// NETWORK 70
P3_FB_Temperature[78](bReset := P3_SystemRUN.bReset, ParTemp := arrTempPar[78], TempCtrl := arrTempCtrl[78]); // FB_Temperature

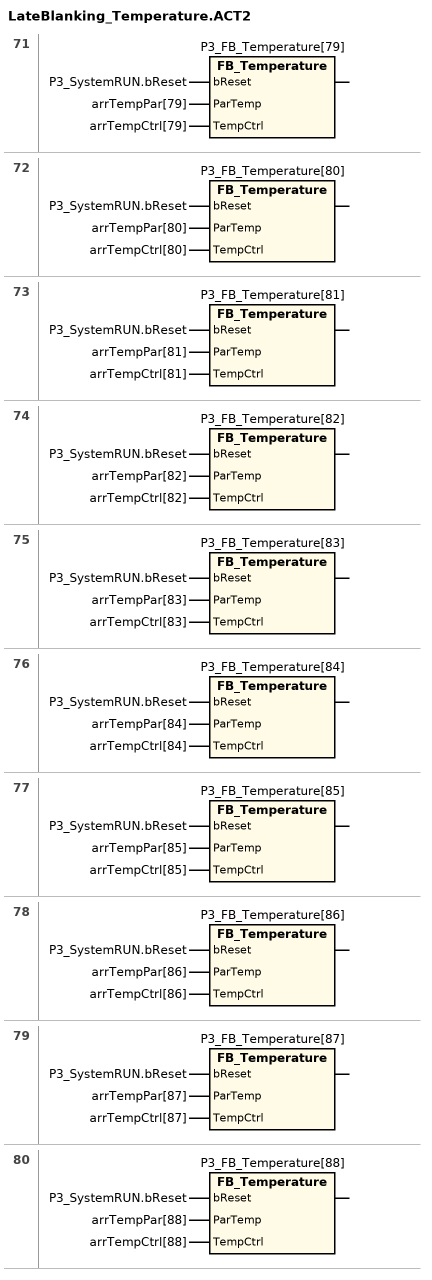
// NETWORK 71
P3_FB_Temperature[79](bReset := P3_SystemRUN.bReset, ParTemp := arrTempPar[79], TempCtrl := arrTempCtrl[79]); // FB_Temperature

// NETWORK 72
P3_FB_Temperature[80](bReset := P3_SystemRUN.bReset, ParTemp := arrTempPar[80], TempCtrl := arrTempCtrl[80]); // FB_Temperature

// NETWORK 73
P3_FB_Temperature[81](bReset := P3_SystemRUN.bReset, ParTemp := arrTempPar[81], TempCtrl := arrTempCtrl[81]); // FB_Temperature

// NETWORK 74
P3_FB_Temperature[82](bReset := P3_SystemRUN.bReset, ParTemp := arrTempPar[82], TempCtrl := arrTempCtrl[82]); // FB_Temperature

// NETWORK 75
P3_FB_Temperature[83](bReset := P3_SystemRUN.bReset, ParTemp := arrTempPar[83], TempCtrl := arrTempCtrl[83]); // FB_Temperature

// NETWORK 76
P3_FB_Temperature[84](bReset := P3_SystemRUN.bReset, ParTemp := arrTempPar[84], TempCtrl := arrTempCtrl[84]); // FB_Temperature

// NETWORK 77
P3_FB_Temperature[85](bReset := P3_SystemRUN.bReset, ParTemp := arrTempPar[85], TempCtrl := arrTempCtrl[85]); // FB_Temperature

// NETWORK 78
P3_FB_Temperature[86](bReset := P3_SystemRUN.bReset, ParTemp := arrTempPar[86], TempCtrl := arrTempCtrl[86]); // FB_Temperature

// NETWORK 79
P3_FB_Temperature[87](bReset := P3_SystemRUN.bReset, ParTemp := arrTempPar[87], TempCtrl := arrTempCtrl[87]); // FB_Temperature

// NETWORK 80
P3_FB_Temperature[88](bReset := P3_SystemRUN.bReset, ParTemp := arrTempPar[88], TempCtrl := arrTempCtrl[88]); // FB_Temperature

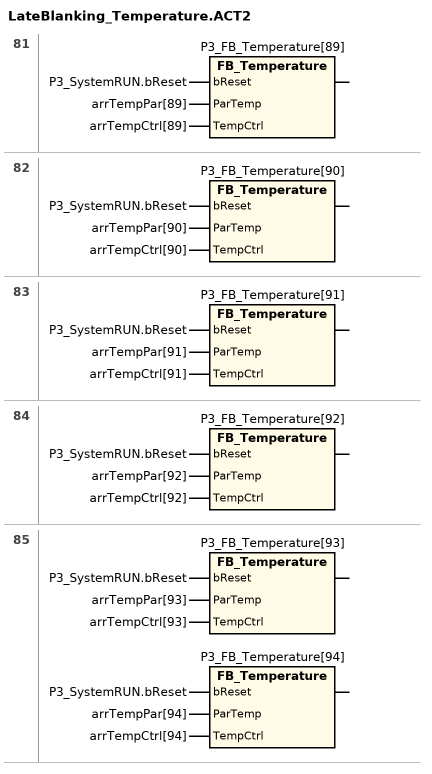
// NETWORK 81
P3_FB_Temperature[89](bReset := P3_SystemRUN.bReset, ParTemp := arrTempPar[89], TempCtrl := arrTempCtrl[89]); // FB_Temperature

// NETWORK 82
P3_FB_Temperature[90](bReset := P3_SystemRUN.bReset, ParTemp := arrTempPar[90], TempCtrl := arrTempCtrl[90]); // FB_Temperature

// NETWORK 83
P3_FB_Temperature[91](bReset := P3_SystemRUN.bReset, ParTemp := arrTempPar[91], TempCtrl := arrTempCtrl[91]); // FB_Temperature

// NETWORK 84
P3_FB_Temperature[92](bReset := P3_SystemRUN.bReset, ParTemp := arrTempPar[92], TempCtrl := arrTempCtrl[92]); // FB_Temperature

// NETWORK 85
P3_FB_Temperature[93](bReset := P3_SystemRUN.bReset, ParTemp := arrTempPar[93], TempCtrl := arrTempCtrl[93]); // FB_Temperature
P3_FB_Temperature[94](bReset := P3_SystemRUN.bReset, ParTemp := arrTempPar[94], TempCtrl := arrTempCtrl[94]); // FB_Temperature
END_ACTION

END_PROGRAM

// ---- P3POUs/POUs/Auxiliary/LateBlanking_Thickness_Test.TcPOU
//测厚测试
PROGRAM LateBlanking_Thickness_Test
VAR
b_Thickness_TON :Tc2_Standard.TON;
b_Thickness_TON2 :TON;
END_VAR

(*IF Permit_Thickness OR Shield[3]  THEN
	CellMemory[CellNo.Thickness].Thickness:=1;
    Thickness_Finish:=TRUE;
	Permit_Thickness:=FALSE;
END_IF*)
b_Thickness_TON(PT:=T#5S);
b_Thickness_TON2(PT:=T#1S);
Thickness_Par_Z:=DINT_TO_REAL(ThicknessPar)/1000;
P3User2_Par.Thick_Cell_Par:=P3User2_Par.Thick_Par - Thickness_Par_Z;
P3User2_Par.Thick_min;//:=Thick_Par-Thick_MN;
P3User2_Par.Thick_max;//:=Thick_Par+Thick_MN;

IF P3_SystemRUN.iMode=1 THEN
CASE  Thickness_Step OF

1://测厚压板打开和测厚托板缩回
	b_Thickness_TON.IN:=FALSE;
	b_Thickness_TON2.IN:=FALSE;
	IF arrCyCtrl[P3CYNo.P3ThicknessSupport].Status.ONState AND  arrCyCtrl[P3CYNo.P3ThicknessMeasuringSwitch].Status.ONState  
		AND arrCyCtrl[P3CYNo.P3ThicknessPressure].Status.OFFState THEN
		Thickness_Step:=30;
	ELSE
		Thickness_Step:=5;
	END_IF
		
5:
	arrCyCtrl[P3CYNo.P3ThicknessSupport].Cmd.bOFF:=TRUE;
	arrCyCtrl[P3CYNo.P3ThicknessPressure].Cmd.bOFF:=TRUE;
	IF 
	   arrCyCtrl[P3CYNo.P3ThicknessSupport].Status.OFFState AND NOT arrCyCtrl[P3CYNo.P3ThicknessSupport].Status.Error2 AND
	   arrCyCtrl[P3CYNo.P3ThicknessPressure].Status.OFFState AND NOT arrCyCtrl[P3CYNo.P3ThicknessPressure].Status.Error2 THEN
	   Thickness_Step:=10;
	END_IF

10://测厚切换气缸伸出
	arrCyCtrl[P3CYNo.P3ThicknessMeasuringSwitch].Cmd.bON:=TRUE;
 
	IF   arrCyCtrl[P3CYNo.P3ThicknessMeasuringSwitch].Status.ONState AND NOT arrCyCtrl[P3CYNo.P3ThicknessMeasuringSwitch].Status.Error1 THEN
		Thickness_Step:=20;
	END_IF

20://测厚托板伸出
	arrCyCtrl[P3CYNo.P3ThicknessSupport].Cmd.bON:=TRUE;
	IF 
	   arrCyCtrl[P3CYNo.P3ThicknessSupport].Status.ONState AND NOT arrCyCtrl[P3CYNo.P3ThicknessSupport].Status.Error1  THEN
	   Thickness_Step:=30;
	END_IF

30://判断是否有允许测厚信号
		IF Permit_Thickness AND NOT Thickness_Finish
		AND arrCyCtrl[P3CYNo.P3ThicknessSupport].Status.ONState AND  arrCyCtrl[P3CYNo.P3ThicknessMeasuringSwitch].Status.ONState  
		AND arrCyCtrl[P3CYNo.P3ThicknessPressure].Status.OFFState THEN
		Thickness_Step:=40;
		ELSIF Step35=100 AND(NOT arrCyCtrl[P3CYNo.P3ThicknessSupport].Status.ONState OR NOT arrCyCtrl[P3CYNo.P3ThicknessMeasuringSwitch].Status.ONState OR NOT arrCyCtrl[P3CYNo.P3ThicknessPressure].Status.OFFState) THEN
		Thickness_Step:=1;
		END_IF 
		
	
40://测厚托板缩回
	arrCyCtrl[P3CYNo.P3ThicknessSupport].Cmd.bOFF:=TRUE;
	IF 	   arrCyCtrl[P3CYNo.P3ThicknessSupport].Status.OFFState AND NOT arrCyCtrl[P3CYNo.P3ThicknessSupport].Status.Error2  THEN
	   			Thickness_Step:=50;
	END_IF  
    
50://测厚切换气缸缩回
	arrCyCtrl[P3CYNo.P3ThicknessMeasuringSwitch].Cmd.bOFF:=TRUE;
 
IF   arrCyCtrl[P3CYNo.P3ThicknessMeasuringSwitch].Status.OFFState AND NOT arrCyCtrl[P3CYNo.P3ThicknessMeasuringSwitch].Status.Error2 THEN
   Thickness_Step:=55;
END_IF

55://检测电芯有无
b_Thickness_TON2.IN:=TRUE;
IF b_Thickness_TON2.Q AND  NOT P3Senser.P3_ThicknessSensor THEN
	P3_Error[55]:=TRUE;//测厚台有记忆无电芯报警
	b_Thickness_TON2.IN:=FALSE;
	Thickness_Step:=100;
ELSE
	b_Thickness_TON2.IN:=FALSE;
	 Thickness_Step:=60;
END_IF

60://测厚压板下压
	b_Thickness_TON.IN:=FALSE;
	arrCyCtrl[P3CYNo.P3ThicknessPressure].Cmd.bON:=TRUE;
		IF    arrCyCtrl[P3CYNo.P3ThicknessPressure].Status.ONState AND NOT arrCyCtrl[P3CYNo.P3ThicknessPressure].Status.Error1 THEN
	   			Thickness_Step:=70;
		END_IF

70:
     b_Thickness_TON.IN:=TRUE;
	 IF b_Thickness_TON.Q THEN
		Thickness_Step:=80;
		b_Thickness_TON.IN:=FALSE;
	END_IF
		
80:
IF 	(P3User2_Par.Thick_Cell_Par<=P3User2_Par.Thick_max AND P3User2_Par.Thick_Cell_Par>=P3User2_Par.Thick_min) OR P3User2_Par.Shield[3] THEN
			CellMemory[CellNo.Thickness].Thickness:=1;
			CellMemory[CellNo.Thickness].Cell_Thickness:=P3User2_Par.Thick_Cell_Par;
			P3par.P3_Thickness_HMIStuas:=1;
			P3par.P3_Thickness_HMIThick:=P3User2_Par.Thick_Cell_Par;
			Thickness_Step:=90;
	ELSIF 	P3User2_Par.Thick_Cell_Par>P3User2_Par.Thick_max OR P3User2_Par.Thick_Cell_Par<P3User2_Par.Thick_min THEN
			CellMemory[CellNo.Thickness].Thickness:=2;
			CellMemory[CellNo.Thickness].Cell_Thickness:=P3User2_Par.Thick_Cell_Par;
			P3par.P3_Thickness_HMIStuas:=2;
			P3par.P3_Thickness_HMIThick:=P3User2_Par.Thick_Cell_Par;		
			Thickness_Step:=90;		
END_IF

90:
		arrCyCtrl[P3CYNo.P3ThicknessPressure].Cmd.bOFF:=TRUE;
		IF    arrCyCtrl[P3CYNo.P3ThicknessPressure].Status.OFFState AND NOT arrCyCtrl[P3CYNo.P3ThicknessPressure].Status.Error2 THEN
	   			Thickness_Step:=100;
		END_IF


100://测厚切换气缸伸出
	arrCyCtrl[P3CYNo.P3ThicknessMeasuringSwitch].Cmd.bON:=TRUE;
 
IF   arrCyCtrl[P3CYNo.P3ThicknessMeasuringSwitch].Status.ONState AND NOT arrCyCtrl[P3CYNo.P3ThicknessMeasuringSwitch].Status.Error1 THEN
   Thickness_Step:=110;
END_IF

110://测厚托板伸出
	arrCyCtrl[P3CYNo.P3ThicknessSupport].Cmd.bON:=TRUE;
	IF 
	   arrCyCtrl[P3CYNo.P3ThicknessSupport].Status.ONState AND NOT arrCyCtrl[P3CYNo.P3ThicknessSupport].Status.Error1  THEN
	   Thickness_Step:=120;
	END_IF


120:
	Permit_Thickness:=FALSE;
	Thickness_Finish:=TRUE;
	 Thickness_Step:=1;
	


		
END_CASE
END_IF

END_PROGRAM

// ---- P3POUs/POUs/Auxiliary/LateBlanking_Weight_Test.TcPOU
//称重测试
PROGRAM LateBlanking_Weight_Test
VAR
	strBetryName: STRING;//文件名

    strBetryName2: STRING;//文件名
	bTest: BOOL;
	AA: UDINT;
	BB: UDINT;
	Weight_cese_1: Weight_cese;
	
	W_ton :Tc2_Standard.TON;
	

	
END_VAR



//称重平台上料
IF NOT Permit_Weigh AND NOT Weigh_Finish THEN
	Permit_WeighRack:=TRUE;
	ELSE
	Permit_WeighRack:=FALSE;
END_IF


W_ton(PT:=T#100MS);
Weight_date();


CASE weight_step OF 
0:
IF Permit_Weigh AND NOT Weigh_Finish AND NOT P3_Error[15]THEN
	weight_step:=10;
END_IF

10:
P3_Weight_gross.Weight_start:=TRUE;
W_ton.IN:=TRUE;
weight_step:=20;

20:
IF( P3_Weight_gross.Weight_finish  AND W_ton.Q)  OR  P3User2_Par.Shield[2]	THEN
	Permit_Weigh:=FALSE;
	Weigh_Finish:=TRUE;
	P3_Weight_gross.Weight_start:=FALSE;
	CellMemory[CellNo.Weight].Cell_weight:=P3_Weight_gross.bweight;
	CellMemory[CellNo.Weight].Weight:=1;
	weight_step:=30;
END_IF

30:
W_ton.IN:=FALSE;
P3_Weight_gross.Weight_finish:=FALSE;
weight_step:=0;
END_CASE






































(*IF bTest THEN
	
 STRING_TO_UTF8(pDstUTF8:=ADR(P3WeightSend.Data) , pSrcSTRING:=ADR(strBetryName) , nDstSize:=INT_TO_UINT( LEN(STR:=strBetryName )+1) );

 AA:=INT_TO_UDINT( LEN(STR:=strBetryName2 )+1);
  BB:=INT_TO_UDINT( LEN(STR:=strBetryName )+1);
 UTF8_TO_STRING(pDstSTRING:=ADR(strBetryName2) , pSrcUTF8:=ADR(P3WeightRec.Data) , nDstSize:=SIZEOF(P3WeightRec.Data) , nDstLen=> AA    );
 bTest:=FALSE;
END_IF*)

ACTION Weight_date:
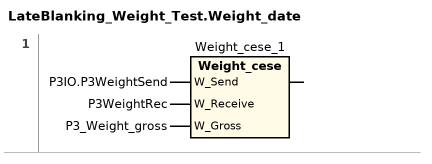
// NETWORK 1
Weight_cese_1(W_Send := P3IO.P3WeightSend, W_Receive := P3WeightRec, W_Gross := P3_Weight_gross); // Weight_cese
END_ACTION

END_PROGRAM

// ---- P3POUs/P3FB/Weight_cese.TcPOU
FUNCTION_BLOCK Weight_cese
VAR_INPUT
	//W_Send :ST_Send;
	
END_VAR
VAR_IN_OUT

	W_Send :ST_SendData;
	W_Receive:ST_ReceiveData;
	W_Gross	:ST_Gross;
END_VAR
VAR_OUTPUT
	
	
END_VAR
VAR
	Step_W_Date :UINT;
	W_TON :ARRAY[1..6] OF Tc2_Standard.TON;
	strBetryName	:STRING;//字符串
	strBetryName2 	:STRING;
	strBetryName3 	:STRING;
	L_R: UDINT;
	L_S: UDINT;
	G_OUT1 	:STRING;
	G_OUT2 	:STRING;
	weight	:REAL;
	weight_Z	:REAL;
	WeightTestAgain :BOOL;
	WeightTestAgainMount :INT;
END_VAR

ACT();
W_TON[1](PT:=T#2S);
W_TON[2](PT:=T#100MS);
W_TON[3](PT:=T#2S);
W_TON[4](PT:=T#100MS);


//初始位称重功能块
IF W_Gross.Init THEN
	Step_W_Date:=0;
	W_Gross.Weight_start:=FALSE;
	W_Gross.Clear_start:=FALSE;
	W_Send.Status.InitRequest:=FALSE;
	W_Send.Status.TransmitRequest:=FALSE;
	W_Gross.error[1]:=FALSE;
	W_Gross.Clear_finish:=FALSE;
	W_Gross.Weight_finish:=FALSE;
	W_Gross.Init:=FALSE;
END_IF





CASE Step_W_Date  OF	
0://称重测试开始
IF W_Gross.Weight_start THEN
	Step_W_Date:=10;
	W_Gross.Weight_finish:=FALSE;
	W_Gross.Weight_start :=FALSE;
	W_Gross.Clear_finish:=FALSE;

ELSIF W_Gross.Clear_start THEN
	Step_W_Date:=1010;
	W_Gross.Clear_finish:=FALSE;
	W_Gross.Clear_start :=FALSE;
	W_Gross.Weight_finish:=FALSE;
END_IF

10://初始化
W_Send.Status.InitRequest:=TRUE;
W_TON[1].IN:=TRUE;
Step_W_Date:=20;

20://如果接收到就
IF W_Receive.Status.InitAccepted THEN
	Step_W_Date:=30;
	W_Send.Status.InitRequest:=FALSE;
	W_TON[1].IN:=FALSE;
END_IF
IF W_TON[1].Q THEN
	W_Send.Status.InitRequest:=FALSE;
	W_Gross.error[1]:=TRUE;
	W_TON[1].IN:=FALSE;
	Step_W_Date:=1111;
END_IF

30:
strBetryName:='Q$R$N';
STRING_TO_UTF8(pDstUTF8:=ADR(W_Send.Data) , pSrcSTRING:=ADR(strBetryName) , nDstSize:=INT_TO_UINT( LEN(STR:=strBetryName )+1));
W_Send.Status.OutputLength:=INT_TO_UINT( LEN(STR:=strBetryName ));
Step_W_Date:=40;

40:
W_Send.Status.TransmitRequest:=TRUE;
IF W_Receive.Status.TransmitDone AND W_Receive.Status.ReceiveRequest AND W_Receive.Status.TotalInputLength>5 THEN
	Step_W_Date:=50;
W_Send.Status.TransmitRequest:=FALSE;
END_IF

50:
L_R:=INT_TO_UDINT( LEN(STR:=strBetryName2 )+1);
UTF8_TO_STRING(pDstSTRING:=ADR(strBetryName2) , pSrcUTF8:=ADR(W_Receive.Data) , nDstSize:=SIZEOF(W_Receive.Data) , nDstLen=> L_R  );
W_TON[2].IN:=TRUE;
IF W_TON[2].Q THEN
Step_W_Date:=60;
W_TON[2].IN:=FALSE;
END_IF

60:
weight_Z:=STRING_TO_REAL(G_OUT2);
IF G_OUT1='+' THEN
	W_Gross.bweight:=weight_Z;
	Step_W_Date:=70;
END_IF
IF G_OUT1='-' THEN
	W_Gross.bweight:=-weight_Z;
	Step_W_Date:=70;
END_IF

70:
IF W_Gross.bweight >=1 OR WeightTestAgain THEN
W_Gross.Weight_finish:=TRUE;
Step_W_Date:=0;
WeightTestAgain:=FALSE;
ELSE
WeightTestAgain:=TRUE;
Step_W_Date:=10;
WeightTestAgainMount:=WeightTestAgainMount+1;
END_IF




1010://初始化
W_Send.Status.InitRequest:=TRUE;
W_TON[3].IN:=TRUE;
Step_W_Date:=1020;

1020://如果接收到就
IF W_Receive.Status.InitAccepted THEN
	Step_W_Date:=1030;
	W_Send.Status.InitRequest:=FALSE;
	W_TON[3].IN:=FALSE;
END_IF
IF W_TON[3].Q THEN
	W_Send.Status.InitRequest:=FALSE;
	W_Gross.error[1]:=TRUE;
	W_TON[3].IN:=FALSE;
	Step_W_Date:=1111;
END_IF

1030:
strBetryName3:='R$R$N';
STRING_TO_UTF8(pDstUTF8:=ADR(W_Send.Data) , pSrcSTRING:=ADR(strBetryName3) , nDstSize:=INT_TO_UINT( LEN(STR:=strBetryName3 )+1   )       );
W_Send.Status.OutputLength:=INT_TO_UINT( LEN(STR:=strBetryName3 ));
Step_W_Date:=1040;

1040:
W_Send.Status.TransmitRequest:=TRUE;
IF W_Receive.Status.TransmitDone  AND W_Receive.Status.ReceiveRequest THEN
	W_Send.Status.TransmitRequest:=FALSE;
	W_Send.Status.ReceiveAccepted:=TRUE;
	Step_W_Date:=1050;
END_IF

1050:
IF NOT W_Receive.Status.ReceiveRequest  THEN
	W_Send.Status.ReceiveAccepted:=FALSE;
	Step_W_Date:=1060;
END_IF

1060:
IF  W_Receive.Status.ReceiveRequest THEN
	W_Gross.Clear_finish:=TRUE;
	Step_W_Date:=0;
END_IF



END_CASE

ACTION ACT:
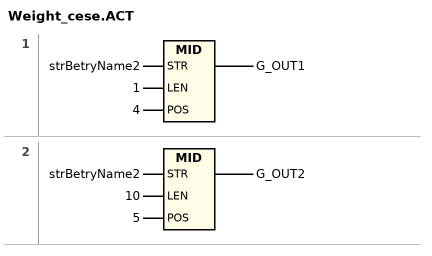
// NETWORK 1
G_OUT1 := MID(STR := strBetryName2, LEN := 1, POS := 4);

// NETWORK 2
G_OUT2 := MID(STR := strBetryName2, LEN := 10, POS := 5);
END_ACTION

END_FUNCTION_BLOCK

// ---- P3POUs/POUs/Auxiliary/LateBlankingCylinderManual.TcPOU
PROGRAM LateBlankingCylinderManual
VAR
    rGluebtn: R_TRIG;//拉胶按钮
	rCutbtn: R_TRIG;//切胶按钮
	rIDGluebtn: R_TRIG;//拉胶按钮
	rIDCutbtn: R_TRIG;//切胶按钮		
END_VAR

//冷压上料夹气缸点动
arrCyCtrl[P3CYNo.P3ColdPressClip].Cmd.ErrorTime:=5;
arrCyCtrl[P3CYNo.P3ColdPressClip].Cmd.iType:=1;
arrCyCtrl[P3CYNo.P3ColdPressClip].Cmd.OffCondition:=TRUE;
arrCyCtrl[P3CYNo.P3ColdPressClip].Cmd.OnCondition:=TRUE;

//冷压麦拉张紧气缸点动
arrCyCtrl[P3CYNo.P3ColdPressTensed].Cmd.ErrorTime:=5;
arrCyCtrl[P3CYNo.P3ColdPressTensed].Cmd.iType:=3;
arrCyCtrl[P3CYNo.P3ColdPressTensed].Cmd.OffCondition:=TRUE;
arrCyCtrl[P3CYNo.P3ColdPressTensed].Cmd.OnCondition:=TRUE;

//烤箱上料夹气缸点动
arrCyCtrl[P3CYNo.P3OvenMoveClip].Cmd.ErrorTime:=5;
arrCyCtrl[P3CYNo.P3OvenMoveClip].Cmd.iType:=1;
arrCyCtrl[P3CYNo.P3OvenMoveClip].Cmd.OffCondition:=TRUE;
arrCyCtrl[P3CYNo.P3OvenMoveClip].Cmd.OnCondition:=TRUE;


//P3 1_1烤箱托板气缸点动
arrCyCtrl[P3CYNo.P3Oven1].Cmd.ErrorTime:=8;
arrCyCtrl[P3CYNo.P3Oven1].Cmd.iType:=1;
IF arrAxisCtrlV2[P3AxisNo.P3_M2_OvenRetracting].Cmd.arrbRealPoint[43] THEN
arrCyCtrl[P3CYNo.P3Oven1].Cmd.OffCondition:=TRUE;
arrCyCtrl[P3CYNo.P3Oven1].Cmd.OnCondition:=TRUE;
ELSE
arrCyCtrl[P3CYNo.P3Oven1].Cmd.OffCondition:=FALSE;
arrCyCtrl[P3CYNo.P3Oven1].Cmd.OnCondition:=FALSE;	
END_IF

//P3 1_2烤箱托板气缸点动
arrCyCtrl[P3CYNo.P3Oven2].Cmd.ErrorTime:=7;
arrCyCtrl[P3CYNo.P3Oven2].Cmd.iType:=1;
IF arrAxisCtrlV2[P3AxisNo.P3_M2_OvenRetracting].Cmd.arrbRealPoint[43] THEN
arrCyCtrl[P3CYNo.P3Oven2].Cmd.OffCondition:=TRUE;
arrCyCtrl[P3CYNo.P3Oven2].Cmd.OnCondition:=TRUE;
ELSE
arrCyCtrl[P3CYNo.P3Oven2].Cmd.OffCondition:=FALSE;
arrCyCtrl[P3CYNo.P3Oven2].Cmd.OnCondition:=FALSE;	
END_IF


//P3 1_3烤箱托板气缸点动
arrCyCtrl[P3CYNo.P3Oven3].Cmd.ErrorTime:=7;
arrCyCtrl[P3CYNo.P3Oven3].Cmd.iType:=1;
IF arrAxisCtrlV2[P3AxisNo.P3_M2_OvenRetracting].Cmd.arrbRealPoint[43]THEN
arrCyCtrl[P3CYNo.P3Oven3].Cmd.OffCondition:=TRUE;
arrCyCtrl[P3CYNo.P3Oven3].Cmd.OnCondition:=TRUE;
ELSE
arrCyCtrl[P3CYNo.P3Oven3].Cmd.OffCondition:=FALSE;
arrCyCtrl[P3CYNo.P3Oven3].Cmd.OnCondition:=FALSE;	
END_IF

//P3 1_4烤箱托板气缸点动
arrCyCtrl[P3CYNo.P3Oven4].Cmd.ErrorTime:=7;
arrCyCtrl[P3CYNo.P3Oven4].Cmd.iType:=1;
IF arrAxisCtrlV2[P3AxisNo.P3_M2_OvenRetracting].Cmd.arrbRealPoint[43] THEN
arrCyCtrl[P3CYNo.P3Oven4].Cmd.OffCondition:=TRUE;
arrCyCtrl[P3CYNo.P3Oven4].Cmd.OnCondition:=TRUE;
ELSE
arrCyCtrl[P3CYNo.P3Oven4].Cmd.OffCondition:=FALSE;
arrCyCtrl[P3CYNo.P3Oven4].Cmd.OnCondition:=FALSE;	
END_IF

//P3 1_5烤箱托板气缸点动
arrCyCtrl[P3CYNo.P3Oven5].Cmd.ErrorTime:=7;
arrCyCtrl[P3CYNo.P3Oven5].Cmd.iType:=1;
IF arrAxisCtrlV2[P3AxisNo.P3_M2_OvenRetracting].Cmd.arrbRealPoint[43]THEN
arrCyCtrl[P3CYNo.P3Oven5].Cmd.OffCondition:=TRUE;
arrCyCtrl[P3CYNo.P3Oven5].Cmd.OnCondition:=TRUE;
ELSE
arrCyCtrl[P3CYNo.P3Oven5].Cmd.OffCondition:=FALSE;
arrCyCtrl[P3CYNo.P3Oven5].Cmd.OnCondition:=FALSE;	
END_IF

//P3 1_6烤箱托板气缸点动
arrCyCtrl[P3CYNo.P3Oven6].Cmd.ErrorTime:=7;
arrCyCtrl[P3CYNo.P3Oven6].Cmd.iType:=1;
IF arrAxisCtrlV2[P3AxisNo.P3_M2_OvenRetracting].Cmd.arrbRealPoint[43] THEN
arrCyCtrl[P3CYNo.P3Oven6].Cmd.OffCondition:=TRUE;
arrCyCtrl[P3CYNo.P3Oven6].Cmd.OnCondition:=TRUE;
ELSE
arrCyCtrl[P3CYNo.P3Oven6].Cmd.OffCondition:=FALSE;
arrCyCtrl[P3CYNo.P3Oven6].Cmd.OnCondition:=FALSE;	
END_IF

//P3 1_7烤箱托板气缸点动
arrCyCtrl[P3CYNo.P3Oven7].Cmd.ErrorTime:=7;
arrCyCtrl[P3CYNo.P3Oven7].Cmd.iType:=1;
IF arrAxisCtrlV2[P3AxisNo.P3_M2_OvenRetracting].Cmd.arrbRealPoint[43] THEN
arrCyCtrl[P3CYNo.P3Oven7].Cmd.OffCondition:=TRUE;
arrCyCtrl[P3CYNo.P3Oven7].Cmd.OnCondition:=TRUE;
ELSE
arrCyCtrl[P3CYNo.P3Oven7].Cmd.OffCondition:=FALSE;
arrCyCtrl[P3CYNo.P3Oven7].Cmd.OnCondition:=FALSE;	
END_IF

//P3 2_1烤箱托板气缸点动
arrCyCtrl[P3CYNo.P3Oven8].Cmd.ErrorTime:=7;
arrCyCtrl[P3CYNo.P3Oven8].Cmd.iType:=1;
IF arrAxisCtrlV2[P3AxisNo.P3_M2_OvenRetracting].Cmd.arrbRealPoint[43] THEN
arrCyCtrl[P3CYNo.P3Oven8].Cmd.OffCondition:=TRUE;
arrCyCtrl[P3CYNo.P3Oven8].Cmd.OnCondition:=TRUE;
ELSE
arrCyCtrl[P3CYNo.P3Oven8].Cmd.OffCondition:=FALSE;
arrCyCtrl[P3CYNo.P3Oven8].Cmd.OnCondition:=FALSE;	
END_IF

//P3 2_2烤箱托板气缸点动
arrCyCtrl[P3CYNo.P3Oven9].Cmd.ErrorTime:=7;
arrCyCtrl[P3CYNo.P3Oven9].Cmd.iType:=1;
IF arrAxisCtrlV2[P3AxisNo.P3_M2_OvenRetracting].Cmd.arrbRealPoint[43] THEN
arrCyCtrl[P3CYNo.P3Oven9].Cmd.OffCondition:=TRUE;
arrCyCtrl[P3CYNo.P3Oven9].Cmd.OnCondition:=TRUE;
ELSE
arrCyCtrl[P3CYNo.P3Oven9].Cmd.OffCondition:=FALSE;
arrCyCtrl[P3CYNo.P3Oven9].Cmd.OnCondition:=FALSE;	
END_IF

//P3 2_3烤箱托板气缸点动
arrCyCtrl[P3CYNo.P3Oven10].Cmd.ErrorTime:=7;
arrCyCtrl[P3CYNo.P3Oven10].Cmd.iType:=1;
IF arrAxisCtrlV2[P3AxisNo.P3_M2_OvenRetracting].Cmd.arrbRealPoint[43] THEN
arrCyCtrl[P3CYNo.P3Oven10].Cmd.OffCondition:=TRUE;
arrCyCtrl[P3CYNo.P3Oven10].Cmd.OnCondition:=TRUE;
ELSE
arrCyCtrl[P3CYNo.P3Oven10].Cmd.OffCondition:=FALSE;
arrCyCtrl[P3CYNo.P3Oven10].Cmd.OnCondition:=FALSE;	
END_IF

//P3 2_4烤箱托板气缸点动
arrCyCtrl[P3CYNo.P3Oven11].Cmd.ErrorTime:=7;
arrCyCtrl[P3CYNo.P3Oven11].Cmd.iType:=1;
IF arrAxisCtrlV2[P3AxisNo.P3_M2_OvenRetracting].Cmd.arrbRealPoint[43] THEN
arrCyCtrl[P3CYNo.P3Oven11].Cmd.OffCondition:=TRUE;
arrCyCtrl[P3CYNo.P3Oven11].Cmd.OnCondition:=TRUE;
ELSE
arrCyCtrl[P3CYNo.P3Oven11].Cmd.OffCondition:=FALSE;
arrCyCtrl[P3CYNo.P3Oven11].Cmd.OnCondition:=FALSE;	
END_IF

//P3 2_5烤箱托板气缸点动
arrCyCtrl[P3CYNo.P3Oven12].Cmd.ErrorTime:=7;
arrCyCtrl[P3CYNo.P3Oven12].Cmd.iType:=1;
IF arrAxisCtrlV2[P3AxisNo.P3_M2_OvenRetracting].Cmd.arrbRealPoint[43] THEN
arrCyCtrl[P3CYNo.P3Oven12].Cmd.OffCondition:=TRUE;
arrCyCtrl[P3CYNo.P3Oven12].Cmd.OnCondition:=TRUE;
ELSE
arrCyCtrl[P3CYNo.P3Oven12].Cmd.OffCondition:=FALSE;
arrCyCtrl[P3CYNo.P3Oven12].Cmd.OnCondition:=FALSE;	
END_IF

//P3 2_6烤箱托板气缸点动
arrCyCtrl[P3CYNo.P3Oven13].Cmd.ErrorTime:=7;
arrCyCtrl[P3CYNo.P3Oven13].Cmd.iType:=1;
IF arrAxisCtrlV2[P3AxisNo.P3_M2_OvenRetracting].Cmd.arrbRealPoint[43] THEN
arrCyCtrl[P3CYNo.P3Oven13].Cmd.OffCondition:=TRUE;
arrCyCtrl[P3CYNo.P3Oven13].Cmd.OnCondition:=TRUE;
ELSE
arrCyCtrl[P3CYNo.P3Oven13].Cmd.OffCondition:=FALSE;
arrCyCtrl[P3CYNo.P3Oven13].Cmd.OnCondition:=FALSE;	
END_IF

//P3 2_7烤箱托板气缸点动
arrCyCtrl[P3CYNo.P3Oven14].Cmd.ErrorTime:=7;
arrCyCtrl[P3CYNo.P3Oven14].Cmd.iType:=1;
IF arrAxisCtrlV2[P3AxisNo.P3_M2_OvenRetracting].Cmd.arrbRealPoint[43] THEN
arrCyCtrl[P3CYNo.P3Oven14].Cmd.OffCondition:=TRUE;
arrCyCtrl[P3CYNo.P3Oven14].Cmd.OnCondition:=TRUE;
ELSE
arrCyCtrl[P3CYNo.P3Oven14].Cmd.OffCondition:=FALSE;
arrCyCtrl[P3CYNo.P3Oven14].Cmd.OnCondition:=FALSE;	
END_IF

//P3 3_1烤箱托板气缸点动
arrCyCtrl[P3CYNo.P3Oven15].Cmd.ErrorTime:=7;
arrCyCtrl[P3CYNo.P3Oven15].Cmd.iType:=1;
IF arrAxisCtrlV2[P3AxisNo.P3_M2_OvenRetracting].Cmd.arrbRealPoint[43] THEN
arrCyCtrl[P3CYNo.P3Oven15].Cmd.OffCondition:=TRUE;
arrCyCtrl[P3CYNo.P3Oven15].Cmd.OnCondition:=TRUE;
ELSE
arrCyCtrl[P3CYNo.P3Oven15].Cmd.OffCondition:=FALSE;
arrCyCtrl[P3CYNo.P3Oven15].Cmd.OnCondition:=FALSE;	
END_IF

//P3 3_2烤箱托板气缸点动
arrCyCtrl[P3CYNo.P3Oven16].Cmd.ErrorTime:=7;
arrCyCtrl[P3CYNo.P3Oven16].Cmd.iType:=1;
IF arrAxisCtrlV2[P3AxisNo.P3_M2_OvenRetracting].Cmd.arrbRealPoint[43] THEN
arrCyCtrl[P3CYNo.P3Oven16].Cmd.OffCondition:=TRUE;
arrCyCtrl[P3CYNo.P3Oven16].Cmd.OnCondition:=TRUE;
ELSE
arrCyCtrl[P3CYNo.P3Oven16].Cmd.OffCondition:=FALSE;
arrCyCtrl[P3CYNo.P3Oven16].Cmd.OnCondition:=FALSE;	
END_IF

//P3 3_3烤箱托板气缸点动
arrCyCtrl[P3CYNo.P3Oven17].Cmd.ErrorTime:=7;
arrCyCtrl[P3CYNo.P3Oven17].Cmd.iType:=1;
IF arrAxisCtrlV2[P3AxisNo.P3_M2_OvenRetracting].Cmd.arrbRealPoint[43] THEN
arrCyCtrl[P3CYNo.P3Oven17].Cmd.OffCondition:=TRUE;
arrCyCtrl[P3CYNo.P3Oven17].Cmd.OnCondition:=TRUE;
ELSE
arrCyCtrl[P3CYNo.P3Oven17].Cmd.OffCondition:=FALSE;
arrCyCtrl[P3CYNo.P3Oven17].Cmd.OnCondition:=FALSE;	
END_IF

//P3 3_4烤箱托板气缸点动
arrCyCtrl[P3CYNo.P3Oven18].Cmd.ErrorTime:=7;
arrCyCtrl[P3CYNo.P3Oven18].Cmd.iType:=1;
IF arrAxisCtrlV2[P3AxisNo.P3_M2_OvenRetracting].Cmd.arrbRealPoint[43] THEN
arrCyCtrl[P3CYNo.P3Oven18].Cmd.OffCondition:=TRUE;
arrCyCtrl[P3CYNo.P3Oven18].Cmd.OnCondition:=TRUE;
ELSE
arrCyCtrl[P3CYNo.P3Oven18].Cmd.OffCondition:=FALSE;
arrCyCtrl[P3CYNo.P3Oven18].Cmd.OnCondition:=FALSE;	
END_IF

//P3 3_5烤箱托板气缸点动
arrCyCtrl[P3CYNo.P3Oven19].Cmd.ErrorTime:=7;
arrCyCtrl[P3CYNo.P3Oven19].Cmd.iType:=1;
IF arrAxisCtrlV2[P3AxisNo.P3_M2_OvenRetracting].Cmd.arrbRealPoint[43] THEN
arrCyCtrl[P3CYNo.P3Oven19].Cmd.OffCondition:=TRUE;
arrCyCtrl[P3CYNo.P3Oven19].Cmd.OnCondition:=TRUE;
ELSE
arrCyCtrl[P3CYNo.P3Oven19].Cmd.OffCondition:=FALSE;
arrCyCtrl[P3CYNo.P3Oven19].Cmd.OnCondition:=FALSE;	
END_IF

//P3 3_6烤箱托板气缸点动
arrCyCtrl[P3CYNo.P3Oven20].Cmd.ErrorTime:=7;
arrCyCtrl[P3CYNo.P3Oven20].Cmd.iType:=1;
IF arrAxisCtrlV2[P3AxisNo.P3_M2_OvenRetracting].Cmd.arrbRealPoint[43] THEN
arrCyCtrl[P3CYNo.P3Oven20].Cmd.OffCondition:=TRUE;
arrCyCtrl[P3CYNo.P3Oven20].Cmd.OnCondition:=TRUE;
ELSE
arrCyCtrl[P3CYNo.P3Oven20].Cmd.OffCondition:=FALSE;
arrCyCtrl[P3CYNo.P3Oven20].Cmd.OnCondition:=FALSE;	
END_IF

//P3 3_7烤箱托板气缸点动
arrCyCtrl[P3CYNo.P3Oven21].Cmd.ErrorTime:=7;
arrCyCtrl[P3CYNo.P3Oven21].Cmd.iType:=1;
IF arrAxisCtrlV2[P3AxisNo.P3_M2_OvenRetracting].Cmd.arrbRealPoint[43] THEN
arrCyCtrl[P3CYNo.P3Oven21].Cmd.OffCondition:=TRUE;
arrCyCtrl[P3CYNo.P3Oven21].Cmd.OnCondition:=TRUE;
ELSE
arrCyCtrl[P3CYNo.P3Oven21].Cmd.OffCondition:=FALSE;
arrCyCtrl[P3CYNo.P3Oven21].Cmd.OnCondition:=FALSE;	
END_IF

//P3 热压麦拉张紧气缸点动
arrCyCtrl[P3CYNo.P3HotPressTensed].Cmd.ErrorTime:=5;
arrCyCtrl[P3CYNo.P3HotPressTensed].Cmd.iType:=3;
arrCyCtrl[P3CYNo.P3HotPressTensed].Cmd.OffCondition:=TRUE;
arrCyCtrl[P3CYNo.P3HotPressTensed].Cmd.OnCondition:=TRUE;

//P3 短路测试夹气缸点动
arrCyCtrl[P3CYNo.P3ShortTest].Cmd.ErrorTime:=5;
arrCyCtrl[P3CYNo.P3ShortTest].Cmd.iType:=1;
arrCyCtrl[P3CYNo.P3ShortTest].Cmd.OffCondition:=TRUE;
arrCyCtrl[P3CYNo.P3ShortTest].Cmd.OnCondition:=TRUE;

//P3 称重上料夹气缸点动
arrCyCtrl[P3CYNo.P3WeightFeedingClamp].Cmd.ErrorTime:=5;
arrCyCtrl[P3CYNo.P3WeightFeedingClamp].Cmd.iType:=1;
arrCyCtrl[P3CYNo.P3WeightFeedingClamp].Cmd.OffCondition:=TRUE;
arrCyCtrl[P3CYNo.P3WeightFeedingClamp].Cmd.OnCondition:=TRUE;

//P3 测厚台切换气缸点动
arrCyCtrl[P3CYNo.P3ThicknessMeasuringSwitch].Cmd.ErrorTime:=5;
arrCyCtrl[P3CYNo.P3ThicknessMeasuringSwitch].Cmd.iType:=1;
//arrCyCtrl[P3CYNo.P3ThicknessMeasuringSwitch].Cmd.OffCondition:=TRUE;
//arrCyCtrl[P3CYNo.P3ThicknessMeasuringSwitch].Cmd.OnCondition:=TRUE;

//P3 测厚台托板气缸点动
arrCyCtrl[P3CYNo.P3ThicknessSupport].Cmd.ErrorTime:=5;
arrCyCtrl[P3CYNo.P3ThicknessSupport].Cmd.iType:=1;
//arrCyCtrl[P3CYNo.P3ThicknessSupport].Cmd.OffCondition:=TRUE;
//arrCyCtrl[P3CYNo.P3ThicknessSupport].Cmd.OnCondition:=TRUE;

//P3 测厚台压板气缸点动
arrCyCtrl[P3CYNo.P3ThicknessPressure].Cmd.ErrorTime:=5;
arrCyCtrl[P3CYNo.P3ThicknessPressure].Cmd.iType:=1;
arrCyCtrl[P3CYNo.P3ThicknessPressure].Cmd.OffCondition:=TRUE;
//arrCyCtrl[P3CYNo.P3ThicknessPressure].Cmd.OnCondition:=TRUE;

//电芯分选夹开合气缸点动
arrCyCtrl[P3CYNo.P3SortClamp].Cmd.ErrorTime:=5;
arrCyCtrl[P3CYNo.P3SortClamp].Cmd.iType:=1;
arrCyCtrl[P3CYNo.P3SortClamp].Cmd.OffCondition:=TRUE;
arrCyCtrl[P3CYNo.P3SortClamp].Cmd.OnCondition:=TRUE;

//电芯分选夹升降气缸点动
arrCyCtrl[P3CYNo.P3SortLifting].Cmd.ErrorTime:=5;
arrCyCtrl[P3CYNo.P3SortLifting].Cmd.iType:=1;
arrCyCtrl[P3CYNo.P3SortLifting].Cmd.OffCondition:=TRUE;
arrCyCtrl[P3CYNo.P3SortLifting].Cmd.OnCondition:=TRUE;

//电芯分选夹旋转气缸点动
arrCyCtrl[P3CYNo.P3SortRotate].Cmd.ErrorTime:=5;
arrCyCtrl[P3CYNo.P3SortRotate].Cmd.iType:=1;
arrCyCtrl[P3CYNo.P3SortRotate].Cmd.OffCondition:=TRUE;
arrCyCtrl[P3CYNo.P3SortRotate].Cmd.OnCondition:=TRUE;

//电芯下料夹开合气缸点动
arrCyCtrl[P3CYNo.P3BlankingClamp].Cmd.ErrorTime:=5;
arrCyCtrl[P3CYNo.P3BlankingClamp].Cmd.iType:=1;
arrCyCtrl[P3CYNo.P3BlankingClamp].Cmd.OffCondition:=TRUE;
arrCyCtrl[P3CYNo.P3BlankingClamp].Cmd.OnCondition:=TRUE;

//P3电芯下料夹升降气缸点动
arrCyCtrl[P3CYNo.P3BlankingLifting].Cmd.ErrorTime:=5;
arrCyCtrl[P3CYNo.P3BlankingLifting].Cmd.iType:=1;
arrCyCtrl[P3CYNo.P3BlankingLifting].Cmd.OffCondition:=TRUE;
arrCyCtrl[P3CYNo.P3BlankingLifting].Cmd.OnCondition:=TRUE;

//P3电芯NG1料盒锁定气缸点动
arrCyCtrl[P3CYNo.P3BoxLock1_NG].Cmd.ErrorTime:=5;
arrCyCtrl[P3CYNo.P3BoxLock1_NG].Cmd.iType:=1;
arrCyCtrl[P3CYNo.P3BoxLock1_NG].Cmd.OffCondition:=TRUE;
arrCyCtrl[P3CYNo.P3BoxLock1_NG].Cmd.OnCondition:=TRUE;

//P3电芯NG2料盒锁定气缸点动
arrCyCtrl[P3CYNo.P3BoxLock2_NG].Cmd.ErrorTime:=5;
arrCyCtrl[P3CYNo.P3BoxLock2_NG].Cmd.iType:=1;
arrCyCtrl[P3CYNo.P3BoxLock2_NG].Cmd.OffCondition:=TRUE;
arrCyCtrl[P3CYNo.P3BoxLock2_NG].Cmd.OnCondition:=TRUE;

//P3电芯NG3料盒锁定气缸点动
arrCyCtrl[P3CYNo.P3BoxLock3_NG].Cmd.ErrorTime:=5;
arrCyCtrl[P3CYNo.P3BoxLock3_NG].Cmd.iType:=1;
arrCyCtrl[P3CYNo.P3BoxLock3_NG].Cmd.OffCondition:=TRUE;
arrCyCtrl[P3CYNo.P3BoxLock3_NG].Cmd.OnCondition:=TRUE;

//电芯压紧气缸
arrCyCtrl[P3CYNo.P3CellPush].Cmd.iType:=2;

//电电芯平移气缸
arrCyCtrl[P3CYNo.P3CellAdvance].Cmd.iType:=1;

//贴胶头夹紧气缸
arrCyCtrl[P3CYNo.P3TapePush].Cmd.iType:=1;

//拉带夹紧气缸
arrCyCtrl[P3CYNo.P3TapePull].Cmd.iType:=1;

//拉带升降气缸
arrCyCtrl[P3CYNo.P3TapeLift].Cmd.iType:=1;

//切胶气缸
arrCyCtrl[P3CYNo.P3TapeCut].Cmd.iType:=1;

//压胶气缸
arrCyCtrl[P3CYNo.P3GluePush].Cmd.iType:=1;

//贴胶缓存气缸
arrCyCtrl[P3CYNo.P3TapeBuffer].Cmd.iType:=1;

//流水线下料旋转气缸
arrCyCtrl[P3CYNo.P3TapeSpin].Cmd.iType:=1;

//贴胶头真空
arrCyCtrl[P3CYNo.P3TapeVacuo].Cmd.iType:=4;


//P3称重上料夹归正气缸
arrCyCtrl[P3CYNo.P3WgightUP].Cmd.iType:=2;

//P3下料分选夹归正气缸
arrCyCtrl[P3CYNo.P3SortPush].Cmd.iType:=2;

//冷压吹气
arrCyCtrl[P3CYNo.P3ColdBlow].Cmd.iType:=4;

//热压吹气
arrCyCtrl[P3CYNo.P3HotBlow].Cmd.iType:=4;

//P3电芯旋转定位气缸 
arrCyCtrl[P3CYNo.P3CellPushSpin].Cmd.iType:=2;

//P3电芯旋转气缸
arrCyCtrl[P3CYNo.P3CellSpin].Cmd.iType:=1;


arrCyCtrl[P3CYNo.P3_GlueExtend].Cmd.iType:=4;//二维码蹬胶气缸蹬出

arrCyCtrl[P3CYNo.P3_GluePress].Cmd.iType:=2;//二维码压胶气缸压紧

arrCyCtrl[P3CYNo.P3_GlueCut].Cmd.iType:=2;//二维码切胶气缸切胶
arrCyCtrl[P3CYNo.P3_GlueCut].Cmd.OffCondition:=TRUE;
IF arrAxisCtrl[P3AxisNo.P3_IDPut].Cmd.arrbRealPoint[1] OR P3_SystemRUN.iMode=1 OR (LateBlanking_Auto1_Stick.CodeStartMark AND P3_SystemRUN.iMode=3) THEN
arrCyCtrl[P3CYNo.P3_GlueCut].Cmd.OnCondition:=TRUE;	
ELSE
arrCyCtrl[P3CYNo.P3_GlueCut].Cmd.OnCondition:=FALSE;	
END_IF


arrCyCtrl[P3CYNo.P3_GluePull].Cmd.iType:=2;//二维码拉胶气缸夹紧

arrCyCtrl[P3CYNo.P3_GlueVacuum].Cmd.iType:=4;//	二维码贴胶吸盘真空






//拉胶气缸手动
rGluebtn(CLK:=P3Press.Gluebtn , Q=> );
IF NOT arrCyCtrl[P3CYNo.P3TapeLift].Status.OFFState AND rGluebtn.Q AND P3_SystemRUN.iMode=3 AND arrAxisCtrl[P3AxisNo.P3_TapeAdvance].Cmd.arrbRealPoint[1]  
  (* LREAL_TO_REAL(arrAxisCtrl[P3AxisNo.P3_TapeAdvance].Status.fActPos) <= (arrAxisPar[P3AxisNo.P3_TapeAdvance].arrTargetPoint[1]+1)*) THEN
	arrCyCtrl[P3CYNo.P3TapeLift].Cmd.bOFF:=TRUE;
ELSIF NOT arrCyCtrl[P3CYNo.P3TapeLift].Status.ONState AND rGluebtn.Q AND P3_SystemRUN.iMode=3 AND arrAxisCtrl[P3AxisNo.P3_TapeAdvance].Cmd.arrbRealPoint[1]  AND
          arrCyCtrl[P3CYNo.P3TapeCut].Status.OFFState  THEN
	arrCyCtrl[P3CYNo.P3TapeLift].Cmd.bON:=TRUE;
END_IF

//切胶气缸手动
rCutbtn(CLK:=P3Press.Cutbtn , Q=> );
IF NOT arrCyCtrl[P3CYNo.P3TapeCut].Status.OFFState AND rCutbtn.Q AND P3_SystemRUN.iMode=3 THEN
	arrCyCtrl[P3CYNo.P3TapeCut].Cmd.bOFF:=TRUE;
ELSIF NOT arrCyCtrl[P3CYNo.P3TapeCut].Status.ONState AND rCutbtn.Q AND P3_SystemRUN.iMode=3 AND
      arrCyCtrl[P3CYNo.P3TapeLift].Status.OFFState THEN
	arrCyCtrl[P3CYNo.P3TapeCut].Cmd.bON:=TRUE;
END_IF
//切胶气缸手动
rIDCutbtn(CLK:=P3Button.IDCutbtn , Q=> );
IF NOT arrCyCtrl[P3CYNo.P3_GlueCut].Status.OFFState AND rIDCutbtn.Q AND P3_SystemRUN.iMode=3 THEN
	arrCyCtrl[P3CYNo.P3_GlueCut].Cmd.bOFF:=TRUE;
ELSIF NOT arrCyCtrl[P3CYNo.P3_GlueCut].Status.ONState AND rIDCutbtn.Q AND P3_SystemRUN.iMode=3 THEN
	arrCyCtrl[P3CYNo.P3_GlueCut].Cmd.bON:=TRUE;
END_IF

END_PROGRAM

// ---- P3POUs/POUs/Auxiliary/LateBlankingMotorManual.TcPOU
PROGRAM LateBlankingMotorManual
VAR
END_VAR

(*//P3_M1冷压上料夹平移点动
IF arrAxisCtrl[P3AxisNo.P3M1_ColdpreLine].Cmd.hmiJog_Fw THEN
arrAxisCtrl[P3AxisNo.P3M1_ColdpreLine].Cmd.bJog_Fw:=TRUE;
ELSE
arrAxisCtrl[P3AxisNo.P3M1_ColdpreLine].Cmd.bJog_Fw:=FALSE;
END_IF
IF arrAxisCtrl[P3AxisNo.P3M1_ColdpreLine].Cmd.hmibJog_Bw THEN
arrAxisCtrl[P3AxisNo.P3M1_ColdpreLine].Cmd.bJog_Bw:=TRUE;
ELSE
arrAxisCtrl[P3AxisNo.P3M1_ColdpreLine].Cmd.bJog_Bw:=FALSE;
END_IF

//P3_M1冷压上料夹进退点动
IF arrAxisCtrl[P3AxisNo.P3M1_ColdpreRetracting].Cmd.hmiJog_Fw THEN
arrAxisCtrl[P3AxisNo.P3M1_ColdpreRetracting].Cmd.bJog_Fw:=TRUE;
ELSE
arrAxisCtrl[P3AxisNo.P3M1_ColdpreRetracting].Cmd.bJog_Fw:=FALSE;
END_IF
IF arrAxisCtrl[P3AxisNo.P3M1_ColdpreRetracting].Cmd.hmibJog_Bw THEN
arrAxisCtrl[P3AxisNo.P3M1_ColdpreRetracting].Cmd.bJog_Bw:=TRUE;
ELSE
arrAxisCtrl[P3AxisNo.P3M1_ColdpreRetracting].Cmd.bJog_Bw:=FALSE;
END_IF

//P3_M1冷压上料夹旋转点动
IF arrAxisCtrl[P3AxisNo.P3M1_ColdpreWhirling].Cmd.hmiJog_Fw THEN
arrAxisCtrl[P3AxisNo.P3M1_ColdpreWhirling].Cmd.bJog_Fw:=TRUE;
ELSE
arrAxisCtrl[P3AxisNo.P3M1_ColdpreWhirling].Cmd.bJog_Fw:=FALSE;
END_IF
IF arrAxisCtrl[P3AxisNo.P3M1_ColdpreWhirling].Cmd.hmibJog_Bw THEN
arrAxisCtrl[P3AxisNo.P3M1_ColdpreWhirling].Cmd.bJog_Bw:=TRUE;
ELSE
arrAxisCtrl[P3AxisNo.P3M1_ColdpreWhirling].Cmd.bJog_Bw:=FALSE;
END_IF

//P3_M1冷压上料夹升降点动
IF arrAxisCtrl[P3AxisNo.P3M1_ColdpreUpDown].Cmd.hmiJog_Fw THEN
arrAxisCtrl[P3AxisNo.P3M1_ColdpreUpDown].Cmd.bJog_Fw:=TRUE;
ELSE
arrAxisCtrl[P3AxisNo.P3M1_ColdpreUpDown].Cmd.bJog_Fw:=FALSE;
END_IF
IF arrAxisCtrl[P3AxisNo.P3M1_ColdpreUpDown].Cmd.hmibJog_Bw THEN
arrAxisCtrl[P3AxisNo.P3M1_ColdpreUpDown].Cmd.bJog_Bw:=TRUE;
ELSE
arrAxisCtrl[P3AxisNo.P3M1_ColdpreUpDown].Cmd.bJog_Bw:=FALSE;
END_IF

//P3_M1冷压托板开合点动
IF arrAxisCtrl[P3AxisNo.P3M1_ColdpreSupPlateLine].Cmd.hmiJog_Fw THEN
arrAxisCtrl[P3AxisNo.P3M1_ColdpreSupPlateLine].Cmd.bJog_Fw:=TRUE;
ELSE
arrAxisCtrl[P3AxisNo.P3M1_ColdpreSupPlateLine].Cmd.bJog_Fw:=FALSE;
END_IF
IF arrAxisCtrl[P3AxisNo.P3M1_ColdpreSupPlateLine].Cmd.hmibJog_Bw THEN
arrAxisCtrl[P3AxisNo.P3M1_ColdpreSupPlateLine].Cmd.bJog_Bw:=TRUE;
ELSE
arrAxisCtrl[P3AxisNo.P3M1_ColdpreSupPlateLine].Cmd.bJog_Bw:=FALSE;
END_IF

//P3_M1冷压驱动点动
IF arrAxisCtrl[P3AxisNo.P3M1_ColdpreActuated].Cmd.hmiJog_Fw THEN
arrAxisCtrl[P3AxisNo.P3M1_ColdpreActuated].Cmd.bJog_Fw:=TRUE;
ELSE
arrAxisCtrl[P3AxisNo.P3M1_ColdpreActuated].Cmd.bJog_Fw:=FALSE;
END_IF
IF arrAxisCtrl[P3AxisNo.P3M1_ColdpreActuated].Cmd.hmibJog_Bw THEN
arrAxisCtrl[P3AxisNo.P3M1_ColdpreActuated].Cmd.bJog_Bw:=TRUE;
ELSE
arrAxisCtrl[P3AxisNo.P3M1_ColdpreActuated].Cmd.bJog_Bw:=FALSE;
END_IF

//P3_M2烤箱上料夹搬运点动
IF arrAxisCtrlV2[P3AxisNo.P3_M2_OvenCarrying].Cmd.hmiJog_Fw THEN
arrAxisCtrlV2[P3AxisNo.P3_M2_OvenCarrying].Cmd.bJog_Fw:=TRUE;
ELSE
arrAxisCtrlV2[P3AxisNo.P3_M2_OvenCarrying].Cmd.bJog_Fw:=FALSE;
END_IF
IF arrAxisCtrlV2[P3AxisNo.P3_M2_OvenCarrying].Cmd.hmibJog_Bw THEN
arrAxisCtrlV2[P3AxisNo.P3_M2_OvenCarrying].Cmd.bJog_Bw:=TRUE;
ELSE
arrAxisCtrlV2[P3AxisNo.P3_M2_OvenCarrying].Cmd.bJog_Bw:=FALSE;
END_IF

//P3_M2烤箱上料夹进退点动
IF arrAxisCtrlV2[P3AxisNo.P3_M2_OvenRetracting].Cmd.hmiJog_Fw THEN
arrAxisCtrlV2[P3AxisNo.P3_M2_OvenRetracting].Cmd.bJog_Fw:=TRUE;
ELSE
arrAxisCtrlV2[P3AxisNo.P3_M2_OvenRetracting].Cmd.bJog_Fw:=FALSE;
END_IF
IF arrAxisCtrlV2[P3AxisNo.P3_M2_OvenRetracting].Cmd.hmibJog_Bw THEN
arrAxisCtrlV2[P3AxisNo.P3_M2_OvenRetracting].Cmd.bJog_Bw:=TRUE;
ELSE
arrAxisCtrlV2[P3AxisNo.P3_M2_OvenRetracting].Cmd.bJog_Bw:=FALSE;
END_IF

//P3_M2烤箱上料夹升降点动
IF arrAxisCtrlV2[P3AxisNo.P3_M2_OvenUpDown].Cmd.hmiJog_Fw THEN
arrAxisCtrlV2[P3AxisNo.P3_M2_OvenUpDown].Cmd.bJog_Fw:=TRUE;
ELSE
arrAxisCtrlV2[P3AxisNo.P3_M2_OvenUpDown].Cmd.bJog_Fw:=FALSE;
END_IF
IF arrAxisCtrlV2[P3AxisNo.P3_M2_OvenUpDown].Cmd.hmibJog_Bw THEN
arrAxisCtrlV2[P3AxisNo.P3_M2_OvenUpDown].Cmd.bJog_Bw:=TRUE;
ELSE
arrAxisCtrlV2[P3AxisNo.P3_M2_OvenUpDown].Cmd.bJog_Bw:=FALSE;
END_IF

//P3_M3热压托板开合点动
IF arrAxisCtrl[P3AxisNo.P3_M3_HotPressingLine].Cmd.hmiJog_Fw THEN
arrAxisCtrl[P3AxisNo.P3_M3_HotPressingLine].Cmd.bJog_Fw:=TRUE;
ELSE
arrAxisCtrl[P3AxisNo.P3_M3_HotPressingLine].Cmd.bJog_Fw:=FALSE;
END_IF
IF arrAxisCtrl[P3AxisNo.P3_M3_HotPressingLine].Cmd.hmibJog_Bw THEN
arrAxisCtrl[P3AxisNo.P3_M3_HotPressingLine].Cmd.bJog_Bw:=TRUE;
ELSE
arrAxisCtrl[P3AxisNo.P3_M3_HotPressingLine].Cmd.bJog_Bw:=FALSE;
END_IF

//P3_M3热压驱动点动
IF arrAxisCtrl[P3AxisNo.P3_M3_HotPressingActuated].Cmd.hmiJog_Fw THEN
arrAxisCtrl[P3AxisNo.P3_M3_HotPressingActuated].Cmd.bJog_Fw:=TRUE;
ELSE
arrAxisCtrl[P3AxisNo.P3_M3_HotPressingActuated].Cmd.bJog_Fw:=FALSE;
END_IF
IF arrAxisCtrl[P3AxisNo.P3_M3_HotPressingActuated].Cmd.hmibJog_Bw THEN
arrAxisCtrl[P3AxisNo.P3_M3_HotPressingActuated].Cmd.bJog_Bw:=TRUE;
ELSE
arrAxisCtrl[P3AxisNo.P3_M3_HotPressingActuated].Cmd.bJog_Bw:=FALSE;
END_IF

//P3_M4称重上料夹平移点动
IF arrAxisCtrl[P3AxisNo.P3_M4_WeighLine].Cmd.hmiJog_Fw THEN
arrAxisCtrl[P3AxisNo.P3_M4_WeighLine].Cmd.bJog_Fw:=TRUE;
ELSE
arrAxisCtrl[P3AxisNo.P3_M4_WeighLine].Cmd.bJog_Fw:=FALSE;
END_IF
IF arrAxisCtrl[P3AxisNo.P3_M4_WeighLine].Cmd.hmibJog_Bw THEN
arrAxisCtrl[P3AxisNo.P3_M4_WeighLine].Cmd.bJog_Bw:=TRUE;
ELSE
arrAxisCtrl[P3AxisNo.P3_M4_WeighLine].Cmd.bJog_Bw:=FALSE;
END_IF

//P3_M4称重上料夹升降点动
IF arrAxisCtrl[P3AxisNo.P3_M4_WeighUpDown].Cmd.hmiJog_Fw THEN
arrAxisCtrl[P3AxisNo.P3_M4_WeighUpDown].Cmd.bJog_Fw:=TRUE;
ELSE
arrAxisCtrl[P3AxisNo.P3_M4_WeighUpDown].Cmd.bJog_Fw:=FALSE;
END_IF
IF arrAxisCtrl[P3AxisNo.P3_M4_WeighUpDown].Cmd.hmibJog_Bw THEN
arrAxisCtrl[P3AxisNo.P3_M4_WeighUpDown].Cmd.bJog_Bw:=TRUE;
ELSE
arrAxisCtrl[P3AxisNo.P3_M4_WeighUpDown].Cmd.bJog_Bw:=FALSE;
END_IF

//P3_M4称重上料夹旋转点动
IF arrAxisCtrl[P3AxisNo.P3_M4_WeighWhirling].Cmd.hmiJog_Fw THEN
arrAxisCtrl[P3AxisNo.P3_M4_WeighWhirling].Cmd.bJog_Fw:=TRUE;
ELSE
arrAxisCtrl[P3AxisNo.P3_M4_WeighWhirling].Cmd.bJog_Fw:=FALSE;
END_IF
IF arrAxisCtrl[P3AxisNo.P3_M4_WeighWhirling].Cmd.hmibJog_Bw THEN
arrAxisCtrl[P3AxisNo.P3_M4_WeighWhirling].Cmd.bJog_Bw:=TRUE;
ELSE
arrAxisCtrl[P3AxisNo.P3_M4_WeighWhirling].Cmd.bJog_Bw:=FALSE;
END_IF

//P3_M4电芯分选夹搬运点动
IF arrAxisCtrl[P3AxisNo.P3_M4_SortingoutCarrying].Cmd.hmiJog_Fw THEN
arrAxisCtrl[P3AxisNo.P3_M4_SortingoutCarrying].Cmd.bJog_Fw:=TRUE;
ELSE
arrAxisCtrl[P3AxisNo.P3_M4_SortingoutCarrying].Cmd.bJog_Fw:=FALSE;
END_IF
IF arrAxisCtrl[P3AxisNo.P3_M4_SortingoutCarrying].Cmd.hmibJog_Bw THEN
arrAxisCtrl[P3AxisNo.P3_M4_SortingoutCarrying].Cmd.bJog_Bw:=TRUE;
ELSE
arrAxisCtrl[P3AxisNo.P3_M4_SortingoutCarrying].Cmd.bJog_Bw:=FALSE;
END_IF

//P3_M4电芯分选夹升降点动
IF arrAxisCtrl[P3AxisNo.P3_M4_SortingoutUpDown].Cmd.hmiJog_Fw THEN
arrAxisCtrl[P3AxisNo.P3_M4_SortingoutUpDown].Cmd.bJog_Fw:=TRUE;
ELSE
arrAxisCtrl[P3AxisNo.P3_M4_SortingoutUpDown].Cmd.bJog_Fw:=FALSE;
END_IF
IF arrAxisCtrl[P3AxisNo.P3_M4_SortingoutUpDown].Cmd.hmibJog_Bw THEN
arrAxisCtrl[P3AxisNo.P3_M4_SortingoutUpDown].Cmd.bJog_Bw:=TRUE;
ELSE
arrAxisCtrl[P3AxisNo.P3_M4_SortingoutUpDown].Cmd.bJog_Bw:=FALSE;
END_IF

//P3_M4电芯下料夹搬运点动
IF arrAxisCtrl[P3AxisNo.P3_M4_OffloadingCarrying].Cmd.hmiJog_Fw THEN
arrAxisCtrl[P3AxisNo.P3_M4_OffloadingCarrying].Cmd.bJog_Fw:=TRUE;
ELSE
arrAxisCtrl[P3AxisNo.P3_M4_OffloadingCarrying].Cmd.bJog_Fw:=FALSE;
END_IF
IF arrAxisCtrl[P3AxisNo.P3_M4_OffloadingCarrying].Cmd.hmibJog_Bw THEN
arrAxisCtrl[P3AxisNo.P3_M4_OffloadingCarrying].Cmd.bJog_Bw:=TRUE;
ELSE
arrAxisCtrl[P3AxisNo.P3_M4_OffloadingCarrying].Cmd.bJog_Bw:=FALSE;
END_IF

//P3_M4电芯下料夹升降点动
IF arrAxisCtrl[P3AxisNo.P3_M4_OffloadingUpDown].Cmd.hmiJog_Fw THEN
arrAxisCtrl[P3AxisNo.P3_M4_OffloadingUpDown].Cmd.bJog_Fw:=TRUE;
ELSE
arrAxisCtrl[P3AxisNo.P3_M4_OffloadingUpDown].Cmd.bJog_Fw:=FALSE;
END_IF
IF arrAxisCtrl[P3AxisNo.P3_M4_OffloadingUpDown].Cmd.hmibJog_Bw THEN
arrAxisCtrl[P3AxisNo.P3_M4_OffloadingUpDown].Cmd.bJog_Bw:=TRUE;
ELSE
arrAxisCtrl[P3AxisNo.P3_M4_OffloadingUpDown].Cmd.bJog_Bw:=FALSE;
END_IF
*)

END_PROGRAM

// ---- P3POUs/POUs/Auxiliary/LateBlanking_Short_Test.TcPOU
PROGRAM LateBlanking_Short_Test
VAR
ShortTest_Start_TON :Tc2_Standard.TON;	
TON_CYShort :Tc2_Standard.TON;
ShortTest_0: ShortTest;
Shortdata_ton :Tc2_Standard.TON;
YS_Short_ton :Tc2_Standard.TON;
FC_ton :Tc2_Standard.TON;
I:INT;
NG_Tim:Tc2_Standard.TON;
OK_Tim:Tc2_Standard.TON;
END_VAR

(*//短路测试//////////////////开通短路测试要删掉
IF Permit_ShortTest OR Shield[1] THEN
	CellMemory[CellNo.Hotpress].ShortTest:=1;
	ShortTest_Finish:=TRUE;
	Permit_ShortTest:=FALSE;
END_IF*)
shortcese();
ShortTest_Start_TON(PT:=T#8S);
TON_CYShort(PT:=T#6S);
Shortdata_ton(PT:=T#200MS);
YS_Short_ton(PT:=T#3.5S);
FC_ton(PT:=T#70MS);



//IF P3_SystemRUN.iMode=1  THEN//OR P3_SystemRUN.iMode=3
CASE Step_Short OF
0:
	TON_CYShort.IN:=FALSE;
	ShortTest_Start_TON.IN:=FALSE;
	arrCyCtrl[P3CYNo.P3ShortTest].Cmd.bOFF:=TRUE;
	P3Senser.P3_ShortTest_Start:=FALSE;
	Shortdata_ton.IN:=FALSE;
	YS_Short_ton.IN:=FALSE;	
	FC_ton.IN:=FALSE;
	I:=0;
	IF arrCyCtrl[P3CYNo.P3ShortTest].Status.OFFState AND NOT arrCyCtrl[P3CYNo.P3ShortTest].Status.Error2   THEN	
		Step_Short:=5;
	END_IF
5:
	IF  NOT ShortTest_Finish AND Permit_ShortTest AND arrAxisCtrl[P3AxisNo.P3_M3_HotPressingLine].Cmd.arrbRealPoint[2]
		 AND arrAxisCtrl[P3AxisNo.P3_M3_HotPressingLine].Status.NoMoving THEN
		Step_Short:=10;
	END_IF
10:
	IF P3User2_Par.Shield[1] THEN
		Step_Short:=0;
		ShortTest_Finish:=TRUE;	
		CellMemory[CellNo.Hotpress].ShortTest:=1;
	ELSIF Permit_ShortTest AND NOT ShortTest_Finish AND NOT P3Senser.P3_ShortTest_Testing AND Pressing[2] THEN
		 Step_Short:=20;
	END_IF 

20:
	TON_CYShort.IN:=TRUE;
    arrCyCtrl[P3CYNo.P3ShortTest].Cmd.bON:=TRUE;	
	IF (arrCyCtrl[P3CYNo.P3ShortTest].Status.ONState AND NOT arrCyCtrl[P3CYNo.P3ShortTest].Status.Error1) OR TON_CYShort.Q THEN	
	Step_Short:=30;
	TON_CYShort.IN:=FALSE;
	END_IF
		
30:
TON_CYShort.IN:=FALSE;
ShortTest_Start_TON.IN:=TRUE;
P3Senser.P3_ShortTest_Start:=TRUE;
IF ShortTest_Start_TON.Q THEN
Step_Short:=40;
ShortTest_Start_TON.IN:=FALSE;
END_IF

40:
ShortTest_Start_TON.IN:=FALSE;
Shortdata_ton.IN:=FALSE;
OK_Tim(IN:=P3Senser.P3_ShortTest_Pass , PT:=T#0.5S , Q=> , ET=> );
NG_Tim(IN:=P3Senser.P3_ShortTest_UpperFall OR P3Senser.P3_ShortTest_LowerFall , PT:=T#0.5S , Q=> , ET=> );
IF NG_Tim.Q THEN
//IF P3Senser.P3_ShortTest_UpperFall OR P3Senser.P3_ShortTest_LowerFall THEN
	CellMemory[CellNo.Hotpress].ShortTest:=2;
	NG_Tim(IN:=FALSE );
	Step_Short:=50;
	SHORT_HOT.bStart:=TRUE;
ELSIF OK_Tim.Q THEN
//ELSIF P3Senser.P3_ShortTest_Pass THEN
	CellMemory[CellNo.Hotpress].ShortTest:=1;
	OK_Tim(IN:=FALSE );
	Step_Short:=50;
	SHORT_HOT.bStart:=TRUE;	
END_IF

50:
Shortdata_ton.IN:=TRUE;
IF Shortdata_ton.Q AND SHORT_HOT.bDone THEN
Step_Short:=60;	
Shortdata_ton.IN:=FALSE;
END_IF

60:
CellMemory[CellNo.Hotpress].Hipot_R:=(SHORT_HOT.Measure);
CellMemory[CellNo.Hotpress].Hipot_Time:=SHORT_HOT.TestTime;
CellMemory[CellNo.Hotpress].Hipot_V:=SHORT_HOT.Voltage;
Step_Short:=70;	

70:
FC_ton.IN:=FALSE;
SHORT_HOT.bDone:=FALSE;
YS_Short_ton.IN:=FALSE;
P3Senser.P3_ShortTest_Start:=FALSE;
arrCyCtrl[P3CYNo.P3ShortTest].Cmd.bOFF:=TRUE;
Step_Short:=73;	

73:
IF ((CellMemory[CellNo.Hotpress].Hipot_R=0 AND CellMemory[CellNo.Hotpress].ShortTest<>2) 
OR CellMemory[CellNo.Hotpress].Hipot_Time=0 OR CellMemory[CellNo.Hotpress].Hipot_V=0) AND I<=3 THEN
	Step_Short:=1000;

	ELSIF ((CellMemory[CellNo.Hotpress].Hipot_R=0 AND CellMemory[CellNo.Hotpress].ShortTest<>2) 
OR CellMemory[CellNo.Hotpress].Hipot_Time=0 OR CellMemory[CellNo.Hotpress].Hipot_V=0) AND I>3 THEN
	Step_Short:=75;
	I:=0;
	CellMemory[CellNo.Hotpress].Hipot_R:=0;
	CellMemory[CellNo.Hotpress].ShortTest:=2;
	ELSE
	Step_Short:=75;
END_IF

(*
75:
	ShortTest_Finish:=TRUE;
	Permit_ShortTest:=FALSE;
	Step_Short:=0;	*)
75:
	IF NOT P3User2_Par.Shield[6] OR CellMemory[CellNo.Hotpress].ShortTest=2 THEN
		ShortTest_Finish:=TRUE;
		Permit_ShortTest:=FALSE;
		Step_Short:=0;	
	ELSE
	   Step_Short:=80;		
	END_IF



80:
YS_Short_ton.IN:=TRUE;	
IF YS_Short_ton.Q THEN
	arrCyCtrl[P3CYNo.P3ShortTest].Cmd.bON:=TRUE;
	YS_Short_ton.IN:=FALSE;
	TON_CYShort.IN:=TRUE;
	Step_Short:=90;
END_IF

90:
	IF TON_CYShort.Q THEN
		ShortTest_Start_TON.IN:=TRUE;
		P3Senser.P3_ShortTest_Start:=TRUE;
		TON_CYShort.IN:=FALSE;
		Step_Short:=100;
	END_IF
	
100:
	IF ShortTest_Start_TON.Q THEN
		Step_Short:=110;
		SHORT_HOT.bStart:=TRUE;
		ShortTest_Start_TON.IN:=FALSE;
	END_IF

110:
  IF P3Senser.P3_ShortTest_Pass AND CellMemory[CellNo.Hotpress].ShortTest=1 THEN
	  CellMemory[CellNo.Hotpress].ShortTest:=1;
	  Step_Short:=120;
	  ELSIF P3Senser.P3_ShortTest_UpperFall OR P3Senser.P3_ShortTest_LowerFall THEN
	   CellMemory[CellNo.Hotpress].ShortTest:=2;
	    Step_Short:=120;
  END_IF

120:
Shortdata_ton.IN:=TRUE;
IF Shortdata_ton.Q AND SHORT_HOT.bDone THEN
Step_Short:=130;	
Shortdata_ton.IN:=FALSE;
END_IF

130:
CellMemory[CellNo.Hotpress].Hipot2_R:=SHORT_HOT.Measure;
Step_Short:=140;	

140:
SHORT_HOT.bDone:=FALSE;
YS_Short_ton.IN:=FALSE;
P3Senser.P3_ShortTest_Start:=FALSE;
arrCyCtrl[P3CYNo.P3ShortTest].Cmd.bOFF:=TRUE;
ShortTest_Finish:=TRUE;
Permit_ShortTest:=FALSE;
Step_Short:=0;	
	
1000:
SHORT_HOT.bStart:=TRUE;
FC_ton.IN:=TRUE;
Step_Short:=1010;

1010:
IF  SHORT_HOT.bDone AND FC_ton.Q THEN
Step_Short:=60;	
FC_ton.IN:=FALSE;
I:=I+1;
END_IF



	
	
END_CASE
//END_IF

ACTION shortcese:
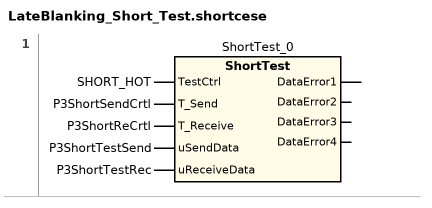
// NETWORK 1
ShortTest_0(
    TestCtrl := SHORT_HOT,
    T_Send := P3ShortSendCrtl,
    T_Receive := P3ShortReCrtl,
    uSendData := P3ShortTestSend,
    uReceiveData := P3ShortTestRec); // ShortTest
END_ACTION

END_PROGRAM

// ---- P3POUs/POUs/Auxiliary/LateBlanking_Scan.TcPOU
PROGRAM LateBlanking_Scan
VAR
	CS_CodeTcp_cold: CS_CodeTcp;
	Cold_step :UINT;
	scan_TON1 :Tc2_Standard.TON;
	Scan_TON :ARRAY[1..7] OF Tc2_Standard.TON;
	Scan_code_Z : R_TRIG;
	I:INT;
END_VAR

//扫码



Saoma();
P3User2_Par.Scan_IP:='192.168.10.26';
Scan_TON[1](PT:=T#1MS);
Scan_TON[2](PT:=T#1MS);
Scan_TON[3](PT:=T#1MS);
Scan_TON[4](PT:=T#100MS);

Scan_code_Z (CLK:=Cold_Scan_code, Q=>);

IF Scan_code_Z.Q AND  Cold_step=0 THEN
	 Cold_step:=10;
END_IF




CASE Cold_step OF
0:
	IF Scan_start AND NOT bCodeError AND NOT bCodeConError AND NOT P3User2_Par.Shield[4] THEN
	 Cold_step:=10;
	 Code_State:=0;
	ELSIF P3User2_Par.Shield[4] THEN
	 Cold_step:=70;
	END_IF
10:
	Scan_TON[1].IN:=FALSE;
	Scan_TON[2].IN:=FALSE;
	Scan_TON[3].IN:=FALSE;
	Cold_step:=20;
	
20:
	bScan_init:=TRUE;
	Scan_TON[1].IN:=TRUE;
	IF Scan_TON[1].Q THEN
		bScan_init:=FALSE;
		Scan_TON[1].IN:=FALSE;
		Cold_step:=30;
	END_IF

30:
	bTcpOpen:=TRUE;
	Scan_TON[2].IN:=TRUE;
	IF Scan_TON[2].Q THEN
		bTcpOpen:=FALSE;
		Scan_TON[2].IN:=FALSE;
		Cold_step:=40;
	END_IF

40:
	IF bTcpOpen_OK THEN
		Cold_step:=50;
	END_IF

50:
	bScan_start:=TRUE;
	Scan_TON[3].IN:=TRUE;
	IF Scan_TON[3].Q THEN
		bScan_start:=FALSE;
		Scan_TON[3].IN:=FALSE;
		Cold_step:=60;
	END_IF
60:
	Scan_TON[4].IN:=TRUE;
	IF 	Scan_TON[4].Q THEN
		Cold_step:=70;
		Scan_TON[4].IN:=FALSE;
	END_IF

70:
IF NOT P3User2_Par.Shield[4] THEN
	IF Code_State=1 AND (strCode<>'') THEN
		CellMemory[CellNo.OvenMoveClip1].Cell_number1:=strCode;
		IF strCode=CellMemory[CellNo.OvenMoveClip1].Cell_number THEN
			CellMemory[CellNo.OvenMoveClip1].ScanCode:=1;
			Scan_start:=FALSE;
			Scan_finish:=TRUE;
			Cold_step:=80;				
			I:=0;
		ELSIF strCode<>CellMemory[CellNo.OvenMoveClip1].Cell_number THEN
			CellMemory[CellNo.OvenMoveClip1].ScanCode:=2;
			P3_Error[79]:=TRUE;//冷压扫码第二次扫码校验NG
			Scan_start:=FALSE;
			Scan_finish:=TRUE;
			Cold_step:=80;
			I:=0;
		END_IF
	ELSIF  Code_State=2 AND I<3 THEN
			Cold_step:=10;
			I:=I+1;		
	ELSIF Code_State=2 AND I>=3 THEN
		CellMemory[CellNo.ColdpressClip].Cell_number1:=strCode;
		CellMemory[CellNo.ColdpressClip].ScanCode:=2;
		P3_Error[16]:=TRUE;//冷压扫码NG报警
		Scan_start:=FALSE;
		Scan_finish:=TRUE;
		Cold_step:=80;
		I:=0;
	END_IF
ELSIF P3User2_Par.Shield[4] THEN
		CellMemory[CellNo.OvenMoveClip1].Cell_number1:='A1234567890ABCDEF';
		CellMemory[CellNo.OvenMoveClip1].ScanCode:=1;
		Scan_start:=FALSE;
		Scan_finish:=TRUE;
		Cold_step:=80;				
		I:=0;
END_IF
80:
	IF NOT Scan_finish THEN
		Cold_step:=0;
	END_IF
END_CASE

ACTION Saoma:
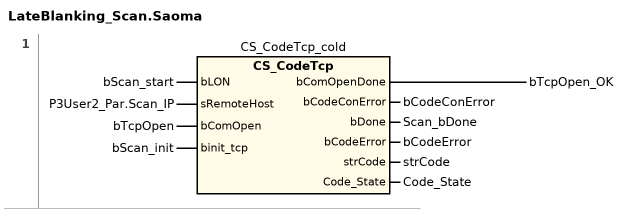
// NETWORK 1
CS_CodeTcp_cold(
    bLON := bScan_start,
    sRemoteHost := P3User2_Par.Scan_IP,
    bComOpen := bTcpOpen,
    binit_tcp := bScan_init,
    bCodeConError => bCodeConError,
    bDone => Scan_bDone,
    bCodeError => bCodeError,
    strCode => strCode,
    Code_State => Code_State); // CS_CodeTcp
bTcpOpen_OK := CS_CodeTcp_cold.bComOpenDone;
END_ACTION

END_PROGRAM

// ---- P3POUs/POUs/Auxiliary/Output_statistics.TcPOU
PROGRAM Output_statistics
VAR
	I:INT;
	DayClear:R_TRIG;
	NightClear:R_TRIG;
	Day_Output_U:UINT;//白班总产量
	Night_Output_U:UINT;//夜班总产量
	Day_Output_NG_U:UINT;// 白班NG数
	Night_Output_NG_U:UINT;// 夜班NG数
	JS_ton1 :ARRAY[0..24] OF ton;//后段运行时间计时
	JS_ton2 :ARRAY[0..24] OF ton;//后段报警时间计时
	His_Hough:R_TRIG;
	P3FB_ProductionDataLocal:FB_ProductionDataLocal;//产能统计
END_VAR



P3FB_ProductionDataLocal(
	NowTimeData:=System.StTime, (*当前系统时间*)
	OutFlag1:=P3_Production.OutFlag1, (*产量计数标志1*)
	OutFlag2:=P3_Production.OutFlag2, (*产量计数标志1*)
	NGFlag:=P3_Production.NGFlag ,(*NG1计数标志*)(*扫码NG*)
	RunFlag:=P3_SystemRUN.iMode=1,(*运行标志*)
	WaitFlag:=P3_SystemRUN.iMode<>1 AND NOT P3_SystemRUN.Alarming ,(*待料标志*)
	AlarmFlag:=P3_SystemRUN.Alarming, (*故障标志*)
	DelDataAMBtn:= P3_Production.HMI_DelDataAMBtn,(*白班数据清除按钮*)//HMI_DayCountZero
	DelDataPMBtn:= P3_Production.HMI_DelDataPMBtn,(*夜班数据清除按钮*)//HMI_NightCountZero
	NowOutTotal=>P3_Production.HMI_TotalCount ,(*当前班次加工总数*)
	NowRate=> P3_Production.HMI_Qualified,(*当前班次良率*)
	OEE=> P3_Production.HMI_OEE,//设备稼动率/稼动率
	NGClearAMBtn:=P3_Production.HMI_NGClearAMBtn,//白班NG类型计数清零
	NGClearPMBtn:=P3_Production.HMI_NGClearPMBtn,//夜班NG类型计数清零
	NowDay:= P3_Production.SaveNowDay,(*数据移位时所保存当前日*)
	NowMonth:=P3_Production.SaveNowMonth ,(*数据移位时所保存当前月*)
	DayHistory:= P3_Production.DayReadDayHistory, (*历史日*)
	MonthHistory:= P3_Production.DayReadMonthHistory,(*历史月*)
	TodayTotal:=P3_Production.HMI_TodayTotal ,(*当天24H生产总数*)
	TodayOK:=P3_Production.HMI_TodayOK , (*当天24H生产OK总数*)
	TodayNG:=P3_Production.HMI_TodayNG , (*当天24H生产NG总数*)
	TodayTotal_AM:= P3_Production.DayCountTotal,(*当天白班生产总数*)
	TodayTotal_PM:=P3_Production.NightCountTotal,(*当天夜班生产总数*)
	TodayRate_AM:= P3_Production.HMI_DayQualified,(*当天白班良率*)
	TodayRate_PM:=P3_Production.HMI_NightQualified ,(*当天夜班良率*)
	TodayOK_AM:=P3_Production.HMI_DayOkCount ,(*当天白班生产OK总数*)
	TodayOK_PM:= P3_Production.HMI_NightOkCount,(*当天夜班生产OK总数*)
	TodayNG_AM:=P3_Production.HMI_DayNgCount ,(*当天白班生产NG总数*)
	TodayNG_PM:=P3_Production.HMI_NightNgCount , (*当天夜班生产NG总数*)
	TodayHour_AM:= P3_Production.HourTimeDayCount,(*当天白班每小时产量ARRAY[8..19 ]*)
	TodayHour_PM:=P3_Production.HourTimeNightCount ,(*当天夜班每小时产量ARRAY[0..23]*)
	TodayNGClass_AM:=P3_Production.NgPerHourDayCount , (*当天白班各类NG数量ARRAY[1..30 ]*)
	TodayNGClass_PM:= P3_Production.NgPerHourNightCount,(*当天夜班各类NG数量ARRAY[1..30 ]*)
	TodayRun_AM:= P3_Production.DayRunTimeTotal,(*当天白班总运行时间合计/分*)
	TodayRun_PM:= P3_Production.NightRunTimeTotal,(*当天夜班总运行时间合计/分*)
	TodayWait_AM:=P3_Production.DayWaitTimeTotal , (*当天白班总待料时间合计/分*)
	TodayWait_PM:=P3_Production.NightWaitTimeTotal , (*当天夜班总待料时间合计/分*)
	TodayAlarm_AM:=P3_Production.DayAlarmTimeTotal ,(*当天白班总报警时间合计/分*)
	TodayAlarm_PM:=P3_Production.NightAlarmTimeTotal, (*当天夜班总报警时间合计/分*)
	
	TodayRun_AMH:=P3_Production.DayRunTime_min,(*当天白班每小时运行时间合计/分*)
	TodayRun_PMH:=P3_Production.NightRunTime_min,(*当天夜班每小时运行时间合计/分*)
	TodayWait_AMH:=P3_Production.DayWaitTime_min,(*当天白班每小时待料时间合计/分*)
	TodayWait_PMH:=P3_Production.NightWaitTime_min,(*当天夜班每小时待料时间合计/分*)
	TodayAlarm_AMH:=P3_Production.DayAlmTime_min,(*当天白班每小时报警时间合计/分*)
	TodayAlarm_PMH:=P3_Production.NightAlmTime_min,(*当天夜班每小时报警时间合计/分*)
	
	HistoryRun_AMH:=P3_Production.HisDayRunTime_min,(*历史每天白班每小时运行时间合计ARRAY[1..7 ]*)
	HistoryRun_PMH:=P3_Production.HisNightRunTime_min,(*历史每天夜班每小时运行时间合计ARRAY[1..7 ]*)
	HistoryWait_AMH:=P3_Production.HisDayWaitTime_min,(*历史每天白班每小时待料时间合计ARRAY[1..7 ]*)
	HistoryWait_PMH:=P3_Production.HisNightWaitTime_min,(*历史每天夜班每小时待料时间合计ARRAY[1..7 ]*)
	HistoryAlarm_AMH:=P3_Production.HisDayAlmTime_min,(*历史每天白班每小时报警时间合计ARRAY[1..7 ]*)
	HistoryAlarm_PMH:=P3_Production.HisNightAlmTime_min,(*历史每天夜班每小时报警时间合计ARRAY[1..7 ]*)
	
	RunCnt_AM:=P3_Production.nDayRunTimeCnt , (*白班运行时间计数*)
	RunCnt_PM:=P3_Production.nNightRunTimeCnt ,(*夜班运行时间计数*)
	WaitCnt_AM:= P3_Production.nDayWaitTimeCnt, (*白班待料时间计数*)
	WaitCnt_PM:=P3_Production.nNightWaitTimeCnt ,(*夜班待料时间计数*)
	AlarmCnt_AM:=P3_Production.nDayAlarmTimeCnt , (*白班报警时间计数*)
	AlarmCnt_PM:= P3_Production.nNightAlarmTimeCnt,(*夜班报警时间计数*)
	
	HistoryTotal:=P3_Production.HMI_HistoryTotal ,(*历史每天24H生产总数ARRAY[1..7 ]*)
	HistoryOK:=P3_Production.HMI_HistoryOK ,(*历史每天24H生产OK总数ARRAY[1..7 ]*)
	HistoryNG:=P3_Production.HMI_HistoryNG , (*历史每天24H生产NG总数ARRAY[1..7 ]*)
	HistoryTotal_AM:=P3_Production.DayCountTotalHistory ,(*历史每天白班生产总数ARRAY[1..7 ]*)
	HistoryTotal_PM:=P3_Production.NightCountTotalHistory ,(*历史每天夜班生产总数ARRAY[1..7 ]*)
	HistoryRate_AM:=P3_Production.HMI_DayQualifiedHistory , (*历史每天白班良率ARRAY[1..7 ]*)
	HistoryRate_PM:=P3_Production.HMI_NightQualifiedHistory,(*历史每天夜班良率ARRAY[1..7 ]*)
	HistoryOK_AM:=P3_Production.HMI_DayOkCountHistory , (*历史每天白班生产OK总数ARRAY[1..7 ]*)
	HistoryOK_PM:=P3_Production.HMI_NightOkCountHistory , (*历史每天夜班生产OK总数ARRAY[1..7 ]*)
	HistoryNG_AM:=P3_Production.HMI_DayNgCountHistory ,(*历史每天白班生产NG总数ARRAY[1..7 ]*)
	HistoryNG_PM:= P3_Production.HMI_NightNgCountHistory,(*历史每天夜班生产NG总数ARRAY[1..7 ]*)
	HistoryHour_AM:=P3_Production.HourTimeDayCountHistory ,(*历史每天白班每小时产量ARRAY[1..7,8..19 ]*)
	HistoryHour_PM:=P3_Production.HourTimeNightCountHistory ,(*历史每天夜班每小时产量ARRAY[1..7,0..23]*)
	HistoryNGClass_AM:= P3_Production.NgPerHourDayCountHistory,(*历史每天白班各类NG数量ARRAY[1..7,1..30 ]*)
	HistoryNGClass_PM:= P3_Production.NgPerHourNightCountHistory,(*历史每天夜班各类NG数量ARRAY[1..7,1..30 ]*)
	HistoryRun_AM:=P3_Production.DayRunTimeTotalHistory , (*历史每天白班总运行时间合计ARRAY[1..7 ]*)
	HistoryRun_PM:= P3_Production.NightRunTimeTotalHistory, (*历史每天夜班总运行时间合计ARRAY[1..7 ]*)
	HistoryWait_AM:= P3_Production.DayWaitTimeTotalHistory,(*历史每天白班总待料时间合计ARRAY[1..7 ]*)
	HistoryWait_PM:= P3_Production.NightWaitTimeTotalHistory, (*历史每天夜班总待料时间合计ARRAY[1..7 ]*)
	HistoryAlarm_AM:= P3_Production.DayAlarmTimeTotalHistory,(*历史每天白班总报警时间合计ARRAY[1..7 ]*)
	HistoryAlarm_PM:= P3_Production.NightAlarmTimeTotalHistory,(*历史每天夜班总报警时间合计ARRAY[1..7 ]*)

	TodayNgHour_Day:=P3_Production.HMINgClassCount_Day,(*白班每种NG类型每小时统计 ,,,NG类型，小时*)
	TodayNgHour_Night:=P3_Production.HMINgClassCount_Night,(*夜班每种NG类型每小时统计 ,,,NG类型，小时*)
	HisTodayNgHour_Day:=P3_Production.HisHMINgClassCount_Day,//l历史白班每小时NG类型统计,,
	HisTodayNgHour_Night:=P3_Production.HisHMINgClassCount_Night,//历史夜班每小时NG类型统计,,
	);

Day_NG.Hough:=REAL_TO_UINT((P2M1_MachCtrl.DT_b.DT_DayHough+P2M2_MachCtrl.DT_b.DT_DayHough+P2M3_MachCtrl.DT_b.DT_DayHough)*100);
Night_NG.Hough:=REAL_TO_UINT((P2M1_MachCtrl.DT_b.DT_NightHough+P2M2_MachCtrl.DT_b.DT_NightHough+P2M3_MachCtrl.DT_b.DT_NightHough)*100);
Day_NG.JDHough:=REAL_TO_UINT((P2M1_MachCtrl.DT_b.DTJD_DayHough+P2M2_MachCtrl.DT_b.DTJD_DayHough+P2M3_MachCtrl.DT_b.DTJD_DayHough)*100);
Night_NG.JDHough:=REAL_TO_UINT((P2M1_MachCtrl.DT_b.DTJD_NightHough+P2M2_MachCtrl.DT_b.DTJD_NightHough+P2M3_MachCtrl.DT_b.DTJD_NightHough)*100);
Day_NG.FirstCheck:=REAL_TO_UINT(P3_Production.NgPerHourDayCount[10]+P3_Production.NgPerHourDayCount[11]+P3_Production.NgPerHourDayCount[12]);
Night_NG.FirstCheck:=REAL_TO_UINT(P3_Production.NgPerHourNightCount[10]+P3_Production.NgPerHourNightCount[11]+P3_Production.NgPerHourNightCount[12]);
//昨日对齐度NG数
His_Hough(CLK:= (System.StTime.wHour=8));
IF His_Hough.Q THEN	
	//白班
	Day_NG.His_Hough:=Day_NG.Hough;
	Day_NG.JDHis_Hough:=Day_NG.JDHough;
	Day_NG.His_FirstCheck:=Day_NG.FirstCheck;
	Day_NG.Hough_DT[1]:=P2M1_MachCtrl.DT_b.DT_DayHough_U; 
	Day_NG.Hough_DT[2]:=P2M2_MachCtrl.DT_b.DT_DayHough_U; 
	Day_NG.Hough_DT[3]:=P2M3_MachCtrl.DT_b.DT_DayHough_U; 
	Day_NG.His_HoughAn[1]:=REAL_TO_UINT(P2M1_MachCtrl.DT_b.DT_DayHoughAn);
	Day_NG.His_HoughAn[2]:=REAL_TO_UINT(P2M2_MachCtrl.DT_b.DT_DayHoughAn);
	Day_NG.His_HoughAn[3]:=REAL_TO_UINT(P2M3_MachCtrl.DT_b.DT_DayHoughAn);
	Day_NG.His_HoughCa[1]:=REAL_TO_UINT(P2M1_MachCtrl.DT_b.DT_DayHoughCa);
	Day_NG.His_HoughCa[2]:=REAL_TO_UINT(P2M2_MachCtrl.DT_b.DT_DayHoughCa);
	Day_NG.His_HoughCa[3]:=REAL_TO_UINT(P2M3_MachCtrl.DT_b.DT_DayHoughCa);
	P2M1_MachCtrl.DT_b.DT_DayHough_U:=0;
	P2M2_MachCtrl.DT_b.DT_DayHough_U:=0;
	P2M3_MachCtrl.DT_b.DT_DayHough_U:=0;
	P2M1_MachCtrl.DT_b.DT_DayHoughAn:=0;
	P2M2_MachCtrl.DT_b.DT_DayHoughAn:=0;
	P2M3_MachCtrl.DT_b.DT_DayHoughAn:=0;
	P2M1_MachCtrl.DT_b.DT_DayHoughCa:=0;
	P2M2_MachCtrl.DT_b.DT_DayHoughCa:=0;
	P2M3_MachCtrl.DT_b.DT_DayHoughCa:=0;
	//夜班
	Night_NG.His_Hough:=Night_NG.Hough;
	Night_NG.JDHis_Hough:=Night_NG.JDHough;
	Night_NG.His_FirstCheck:=Night_NG.FirstCheck;
	Night_NG.Hough_DT[1]:=P2M1_MachCtrl.DT_b.DT_NightHough_U; 
	Night_NG.Hough_DT[2]:=P2M2_MachCtrl.DT_b.DT_NightHough_U; 
	Night_NG.Hough_DT[3]:=P2M3_MachCtrl.DT_b.DT_NightHough_U; 
	Night_NG.His_HoughAn[1]:=REAL_TO_UINT(P2M1_MachCtrl.DT_b.DT_NightHoughAn);
	Night_NG.His_HoughAn[2]:=REAL_TO_UINT(P2M2_MachCtrl.DT_b.DT_NightHoughAn);
	Night_NG.His_HoughAn[3]:=REAL_TO_UINT(P2M3_MachCtrl.DT_b.DT_NightHoughAn);
	Night_NG.His_HoughCa[1]:=REAL_TO_UINT(P2M1_MachCtrl.DT_b.DT_NightHoughCa);
	Night_NG.His_HoughCa[2]:=REAL_TO_UINT(P2M2_MachCtrl.DT_b.DT_NightHoughCa);
	Night_NG.His_HoughCa[3]:=REAL_TO_UINT(P2M3_MachCtrl.DT_b.DT_NightHoughCa);
	P2M1_MachCtrl.DT_b.DT_NightHough_U:=0;
	P2M2_MachCtrl.DT_b.DT_NightHough_U:=0;
	P2M3_MachCtrl.DT_b.DT_NightHough_U:=0;
	P2M1_MachCtrl.DT_b.DT_NightHoughAn:=0;
	P2M2_MachCtrl.DT_b.DT_NightHoughAn:=0;
	P2M3_MachCtrl.DT_b.DT_NightHoughAn:=0;
	P2M1_MachCtrl.DT_b.DT_NightHoughCa:=0;
	P2M2_MachCtrl.DT_b.DT_NightHoughCa:=0;
	P2M3_MachCtrl.DT_b.DT_NightHoughCa:=0;
END_IF

IF system.stTime.wHour >=8 AND system.stTime.wHour <20 THEN
  P3_Production.NgPerHourDayCount[13]:=(MTD_Mes1.rExcelRate[0]+MTD_Mes1.rExcelRate[15])/(P2M1_Par.stDT_date.An_Quantity(*+P2M1_Par.stDT_date.Ca_Quantity*));
 // P3_Production.NgPerHourDayCount[14]:=(MTD_Mes1.rExcelRate[27]+MTD_Mes1.rExcelRate[41])/P2M1_Par.stDT_date.Ca_Quantity;	
  P3_Production.NgPerHourDayCount[15]:=UDINT_TO_REAL(P2M1_Par.stDT_date.An_Rectifydev_DayNG+P2M2_Par.stDT_date.An_Rectifydev_DayNG+P2M3_Par.stDT_date.An_Rectifydev_DayNG)/P2M1_Par.stDT_date.An_Quantity;  
//  P3_Production.NgPerHourDayCount[16]:=UDINT_TO_REAL(P2M1_Par.stDT_date.Ca_Rectifydev_DayNG+P2M2_Par.stDT_date.Ca_Rectifydev_DayNG+P2M3_Par.stDT_date.Ca_Rectifydev_DayNG)/P2M1_Par.stDT_date.Ca_Quantity;  
  P3_Production.NgPerHourDayCount[17]:=(P2M1_MachCtrl.DT_b.DT_DayHoughAn+P2M2_MachCtrl.DT_b.DT_DayHoughAn+P2M3_MachCtrl.DT_b.DT_DayHoughAn)/P2M1_Par.stDT_date.An_Quantity;
END_IF  

IF system.stTime.wHour >=20 OR system.stTime.wHour<8 THEN
  P3_Production.NgPerHourNightCount[13]:=(MTD_Mes1.rExcelRate[0]+MTD_Mes1.rExcelRate[15])/(P2M1_Par.stDT_date.An_Quantity(*+P2M1_Par.stDT_date.Ca_Quantity*));
//  P3_Production.NgPerHourNightCount[14]:=(MTD_Mes1.rExcelRate[27]+MTD_Mes1.rExcelRate[41])/P2M1_Par.stDT_date.Ca_Quantity;	
  P3_Production.NgPerHourNightCount[15]:=UDINT_TO_REAL(P2M1_Par.stDT_date.An_Rectifydev_NightNG+P2M2_Par.stDT_date.An_Rectifydev_NightNG+P2M3_Par.stDT_date.An_Rectifydev_NightNG)/P2M1_Par.stDT_date.An_Quantity;
//  P3_Production.NgPerHourNightCount[16]:=UDINT_TO_REAL(P2M1_Par.stDT_date.Ca_Rectifydev_NightNG+P2M2_Par.stDT_date.Ca_Rectifydev_NightNG+P2M3_Par.stDT_date.Ca_Rectifydev_NightNG)/P2M1_Par.stDT_date.Ca_Quantity;
  P3_Production.NgPerHourNightCount[17]:=(P2M1_MachCtrl.DT_b.DT_NightHoughAn+P2M2_MachCtrl.DT_b.DT_NightHoughAn+P2M3_MachCtrl.DT_b.DT_NightHoughAn)/P2M1_Par.stDT_date.An_Quantity;
END_IF  

//运行时间统计
P3TimeData(
	Alm:= b_Alarm[4] , 
	Wait:=P3_SystemRUN.iMode=3 AND NOT b_Alarm[4] , 
	Run:=P3_SystemRUN.iMode=1 , 
	XL_Wait:=(Step36=1910 OR Step36=1917 ) AND P3_SystemRUN.iMode=1  , 
	Query:=HDQuery, 
	date1:=HDdate , 	
	STTimedata=> );


(*
//产量统计
CASE Output_step OF
100:
		IF CellMemory[CellNo.Thickness].ScanCode<>1  AND Thickness_Finish THEN//踢扫码NG料
				P3_Production.OutFlag1:=TRUE;
				P3_Production.NGFlag[1]:=TRUE;//踢扫码NG料
		ELSIF  CellMemory[CellNo.Thickness].ShortTest<>1 AND Thickness_Finish THEN//踢短路NG料
				P3_Production.OutFlag1:=TRUE;
				P3_Production.NGFlag[2]:=TRUE;//踢短路NG料
		ELSIF CellMemory[CellNo.Thickness].Weight<>1 AND Thickness_Finish THEN//踢称重NG料
				P3_Production.OutFlag1:=TRUE;
				P3_Production.NGFlag[3]:=TRUE;//踢称重NG料
		ELSIF Thickness_Finish AND CellMemory[CellNo.Thickness].Thickness<>1 THEN//测厚NG料
				P3_Production.OutFlag1:=TRUE;
				P3_Production.NGFlag[4]:=TRUE;//测厚NG料
		ELSIF ( NOT CellMemory[CellNo.Thickness].Cell_cold_result OR NOT CellMemory[CellNo.Thickness].Cell_cold_result1 OR NOT CellMemory[CellNo.Thickness].Cell_cold_result2)  AND Thickness_Finish THEN// (NOT CellMemory[CellNo.Thickness].Cell_cold_result OR NOT CellMemory[CellNo.Thickness].Cell_cold_result1 OR
				P3_Production.OutFlag1:=TRUE;
				P3_Production.NGFlag[5]:=TRUE;	//MES卡站NG
		ELSIF Thickness_Finish AND (CellMemory[CellNo.Thickness].ShortTest=1 OR P3User2_Par.Shield[1])  AND (CellMemory[CellNo.Thickness].Weight=1 OR P3User2_Par.Shield[2] ) AND (CellMemory[CellNo.Thickness].Thickness=1 OR P3User2_Par.Shield[3]) THEN
				P3_Production.OutFlag1:=TRUE;//总数
		END_IF
		Output_step:=666;
END_CASE*)








(*
I:=HMI_Hour;


CASE Output_step OF
100://白班、夜班产量统计
IF HMI_Hour>=8 AND HMI_Hour<20 THEN//白班产量
	Day_Output_U:=Day_Output_U+1;
	Day_Output:=(Day_Output_U*100)+Day_NG.Hough;//因触摸屏加了两位小数点，放大100倍
	Output_step:=200;
END_IF
IF (HMI_Hour>=0 AND HMI_Hour<8) OR  (HMI_Hour>=20 AND HMI_Hour<=23) THEN//夜班产量
	Night_Output_U:=Night_Output_U+1;
	Night_Output:=(Night_Output_U*100)+Night_NG.Hough;//因触摸屏加了两位小数点，放大100倍
	Output_step:=200;
END_IF



200://时段产量
	Time_Output[I]:=Time_Output[I]+1;
	Output_step:=300;	

300:
IF HMI_Hour>=8 AND HMI_Hour<20 THEN
		IF CellMemory[CellNo.Thickness].DT_station_No=P2M1_MachCtrl.DT_b.DT_No AND CellMemory[CellNo.Thickness].Hough=2  AND Thickness_Finish THEN
				//	Day_Output_NG:=Day_Output_NG+1;
				//	Day_NG.Hough:=Day_NG.Hough+1;
				//	Day_NG.Hough_DT[1]:=Day_NG.Hough_DT[1]+1;
				Output_step:=1006;
		ELSIF CellMemory[CellNo.Thickness].DT_station_No=P2M2_MachCtrl.DT_b.DT_No AND CellMemory[CellNo.Thickness].Hough=2  AND Thickness_Finish THEN
				//	Day_Output_NG:=Day_Output_NG+1;
				//	Day_NG.Hough:=Day_NG.Hough+1;
				//	Day_NG.Hough_DT[2]:=Day_NG.Hough_DT[2]+1;
				Output_step:=1006;
		ELSIF CellMemory[CellNo.Thickness].DT_station_No=P2M3_MachCtrl.DT_b.DT_No AND CellMemory[CellNo.Thickness].Hough=2  AND Thickness_Finish THEN
				//	Day_Output_NG:=Day_Output_NG+1;
				//	Day_NG.Hough:=Day_NG.Hough+1;
				//	Day_NG.Hough_DT[3]:=Day_NG.Hough_DT[3]+1;
				Output_step:=1006;
		ELSIF CellMemory[CellNo.Thickness].ScanCode<>1  AND Thickness_Finish THEN//踢扫码NG料
				Day_Output_NG_U:=Day_Output_NG_U+1;
				Day_NG.ScanCode:=Day_NG.ScanCode+1;
				Output_step:=1006;
		ELSIF  CellMemory[CellNo.Thickness].ShortTest<>1 AND Thickness_Finish THEN//踢短路NG料
				Day_Output_NG_U:=Day_Output_NG_U+1;
				Day_NG.ShortTest:=Day_NG.ShortTest+1;
				Output_step:=1006;
		ELSIF CellMemory[CellNo.Thickness].Weight<>1 AND Thickness_Finish THEN//踢称重NG料
				Day_Output_NG_U:=Day_Output_NG_U+1;
				Day_NG.Weight:=Day_NG.Weight+1;
				Output_step:=1006; 
		ELSIF Thickness_Finish AND CellMemory[CellNo.Thickness].Thickness<>1 THEN//测厚NG料
				Day_Output_NG_U:=Day_Output_NG_U+1;
				Day_NG.Thickness:=Day_NG.Thickness+1;
				Output_step:=1006;
		ELSIF (NOT CellMemory[CellNo.Thickness].Cell_cold_result OR NOT CellMemory[CellNo.Thickness].Cell_cold_result1 OR NOT CellMemory[CellNo.Thickness].Cell_cold_result2 ) AND Thickness_Finish THEN
				Day_Output_NG_U:=Day_Output_NG_U+1;
				Day_NG.MES:=Day_NG.MES+1;
				Output_step:=1006;	
		ELSIF Thickness_Finish AND (CellMemory[CellNo.Thickness].ShortTest=1 OR P3User2_Par.Shield[1])  AND (CellMemory[CellNo.Thickness].Weight=1 OR P3User2_Par.Shield[2] ) AND (CellMemory[CellNo.Thickness].Thickness=1 OR P3User2_Par.Shield[3]) THEN
				Day_Output_OK:=Day_Output_OK+1;
				Output_step:=1006;
		END_IF
ELSIF (HMI_Hour>=0 AND HMI_Hour<8) OR  (HMI_Hour>=20 AND HMI_Hour<=23) THEN
		IF CellMemory[CellNo.Thickness].DT_station_No=P2M1_MachCtrl.DT_b.DT_No AND CellMemory[CellNo.Thickness].Hough=2  AND Thickness_Finish THEN
				//	Night_Output_NG:=Night_Output_NG+1;
				//	Night_NG.Hough:=Night_NG.Hough+1;
				//	Night_NG.Hough_DT[1]:=Night_NG.Hough_DT[1]+1;
				Output_step:=2006;
		ELSIF CellMemory[CellNo.Thickness].DT_station_No=P2M2_MachCtrl.DT_b.DT_No AND  CellMemory[CellNo.Thickness].Hough=2  AND Thickness_Finish THEN
				//	Night_Output_NG:=Night_Output_NG+1;
				//	Night_NG.Hough:=Night_NG.Hough+1;
				//	Night_NG.Hough_DT[2]:=Night_NG.Hough_DT[2]+1;
				Output_step:=2006;
		ELSIF CellMemory[CellNo.Thickness].DT_station_No=P2M3_MachCtrl.DT_b.DT_No AND  CellMemory[CellNo.Thickness].Hough=2  AND Thickness_Finish THEN
				//	Night_Output_NG:=Night_Output_NG+1;
				//	Night_NG.Hough:=Night_NG.Hough+1;
				//	Night_NG.Hough_DT[3]:=Night_NG.Hough_DT[3]+1;
				Output_step:=2006;
		ELSIF CellMemory[CellNo.Thickness].ScanCode<>1  AND Thickness_Finish THEN//踢扫码NG料
				Night_Output_NG_U:=Night_Output_NG_U+1;
				Night_NG.ScanCode:=Night_NG.ScanCode+1;
				Output_step:=2006;
		ELSIF  CellMemory[CellNo.Thickness].ShortTest<>1 AND Thickness_Finish THEN//踢短路NG料
				Night_Output_NG_U:=Night_Output_NG_U+1;
				Night_NG.ShortTest:=Night_NG.ShortTest+1;
				Output_step:=2006;
		ELSIF CellMemory[CellNo.Thickness].Weight<>1 AND Thickness_Finish THEN//踢称重和测厚NG料
				Night_Output_NG_U:=Night_Output_NG_U+1;
				Night_NG.Weight:=Night_NG.Weight+1;
				Output_step:=2006; 
		ELSIF Thickness_Finish AND CellMemory[CellNo.Thickness].Thickness<>1 THEN
				Night_Output_NG_U:=Night_Output_NG_U+1;
				Night_NG.Thickness:=Night_NG.Thickness+1;
				Output_step:=2006;
		ELSIF (NOT CellMemory[CellNo.Thickness].Cell_cold_result OR NOT CellMemory[CellNo.Thickness].Cell_cold_result1 OR NOT CellMemory[CellNo.Thickness].Cell_cold_result2 ) AND Thickness_Finish THEN
				Night_Output_NG_U:=Night_Output_NG_U+1;
				Night_NG.MES:=Night_NG.MES+1;
				Output_step:=2006;	
		ELSIF Thickness_Finish AND (CellMemory[CellNo.Thickness].ShortTest=1 OR P3User2_Par.Shield[1])  AND (CellMemory[CellNo.Thickness].Weight=1 OR P3User2_Par.Shield[2] ) AND (CellMemory[CellNo.Thickness].Thickness=1 OR P3User2_Par.Shield[3]) THEN
				Night_Output_OK:=Night_Output_OK+1;
				Output_step:=2006;
		END_IF
END_IF



END_CASE

Day_Output_NG:=(Day_Output_NG_U*100)+Day_NG.Hough;//因触摸屏加了两位小数点，放大100倍
Night_Output_NG:=(Night_Output_NG_U*100)+Night_NG.Hough;//因触摸屏加了两位小数点，放大100倍

IF Day_Output<>0 THEN 
Day_Yield:=UINT_TO_REAL(Day_Output_OK)/((UINT_TO_REAL(Day_Output))/100);
END_IF

IF Night_Output<>0 THEN
Night_Yield:=UINT_TO_REAL(Night_Output_OK)/((UINT_TO_REAL(Night_Output))/100);	
END_IF





DayClear(CLK:=(HMI_Hour=8 AND HMI_Minute=0 AND HMI_Second=0 ) , Q=> );
NightClear(CLK:=(HMI_Hour=20 AND HMI_Minute=0 AND HMI_Second=0) , Q=> );



IF Day_Clear OR  DayClear.Q  THEN
	Time_Output[8]:=0;
	Time_Output[9]:=0;
	Time_Output[10]:=0;
	Time_Output[11]:=0;
	Time_Output[12]:=0;
	Time_Output[13]:=0;
	Time_Output[14]:=0;
	Time_Output[15]:=0;
	Time_Output[16]:=0;
	Time_Output[17]:=0;
	Time_Output[18]:=0;
	Time_Output[19]:=0;
	Day_Output_NG:=0;
	Day_Output_OK:=0;
	Day_Output:=0;
	Day_Output_U:=0;
	Day_Output_NG_U:=0;
	Day_Yield:=0;
	MEMSET(ADR(Day_NG),0,SIZEOF(Day_NG));
END_IF

IF Night_Clear OR NightClear.Q THEN
	Time_Output[0]:=0;
	Time_Output[1]:=0;
	Time_Output[2]:=0;
	Time_Output[3]:=0;
	Time_Output[4]:=0;
	Time_Output[5]:=0;
	Time_Output[6]:=0;
	Time_Output[7]:=0;
	Time_Output[20]:=0;
	Time_Output[21]:=0;
	Time_Output[22]:=0;
	Time_Output[23]:=0;
	Night_Output_NG:=0;
	Night_Output_OK:=0;
	Night_Output:=0;
	Night_Output_U:=0;
	Night_Output_NG_U:=0;
	Night_Yield:=0;
	MEMSET(ADR(Night_NG),0,SIZEOF(Night_NG));
END_IF


JS_ton1[0](PT:=T#1000MS);
JS_ton2[0](PT:=T#1000MS);
//1000ms计数一次 次数变量要断电保持
IF HMI_Hour=0 THEN//0:00-1:00
JS_ton1[0].IN:=(b_Alarm[4] AND NOT JS_ton1[0].Q);
 
IF JS_ton1[0].Q THEN
	Alarm_CS[0]:=Alarm_CS[0]+1;
END_IF
JS_ton2[0].IN:=(P3_SystemRUN.iMode=1 AND NOT JS_ton2[0].Q );

IF JS_ton2[0].Q THEN
	Auto_CS[0]:=Auto_CS[0]+1;	
END_IF
Manul_CS[0]:=3600-(Alarm_CS[0]+Auto_CS[0]);
END_IF

JS_ton1[1](PT:=T#1000MS);
JS_ton2[1](PT:=T#1000MS);
IF HMI_Hour=1 THEN//1:00-2:00
JS_ton1[1].IN:=(b_Alarm[4] AND NOT JS_ton1[1].Q);
 
IF JS_ton1[1].Q THEN
	Alarm_CS[1]:=Alarm_CS[1]+1;
END_IF
JS_ton2[1].IN:=(P3_SystemRUN.iMode=1 AND NOT JS_ton2[1].Q );

IF JS_ton2[1].Q THEN
	Auto_CS[1]:=Auto_CS[1]+1;
	
END_IF
Manul_CS[1]:=3600-(Alarm_CS[1]+Auto_CS[1]);
END_IF


JS_ton1[2](PT:=T#1000MS);
JS_ton2[2](PT:=T#1000MS);
IF HMI_Hour=2 THEN//2:00-3:00
JS_ton1[2].IN:=(b_Alarm[4] AND NOT JS_ton1[2].Q);
 
IF JS_ton1[2].Q THEN
	Alarm_CS[2]:=Alarm_CS[2]+1;
END_IF
JS_ton2[2].IN:=(P3_SystemRUN.iMode=1 AND NOT JS_ton2[2].Q );

IF JS_ton2[2].Q THEN
	Auto_CS[2]:=Auto_CS[2]+1;
	
END_IF

Manul_CS[2]:=3600-(Alarm_CS[2]+Auto_CS[2]);

END_IF


JS_ton1[3](PT:=T#1000MS);
JS_ton2[3](PT:=T#1000MS);
IF HMI_Hour=3 THEN//3:00-4:00
JS_ton1[3].IN:=(b_Alarm[4] AND NOT JS_ton1[3].Q);
 
IF JS_ton1[3].Q THEN
	Alarm_CS[3]:=Alarm_CS[3]+1;
END_IF
JS_ton2[3].IN:=(P3_SystemRUN.iMode=1 AND NOT JS_ton2[3].Q );

IF JS_ton2[3].Q THEN
	Auto_CS[3]:=Auto_CS[3]+1;
	
END_IF

Manul_CS[3]:=3600-(Alarm_CS[3]+Auto_CS[3]);

END_IF


JS_ton1[4](PT:=T#1000MS);
JS_ton2[4](PT:=T#1000MS);
IF HMI_Hour=4 THEN//4:00-5:00
JS_ton1[4].IN:=(b_Alarm[4] AND NOT JS_ton1[4].Q);
 
IF JS_ton1[4].Q THEN
	Alarm_CS[4]:=Alarm_CS[4]+1;
END_IF
JS_ton2[4].IN:=(P3_SystemRUN.iMode=1 AND NOT JS_ton2[4].Q );

IF JS_ton2[4].Q THEN
	Auto_CS[4]:=Auto_CS[4]+1;
	
END_IF

Manul_CS[4]:=3600-(Alarm_CS[4]+Auto_CS[4]);

END_IF


JS_ton1[5](PT:=T#1000MS);
JS_ton2[5](PT:=T#1000MS);
IF HMI_Hour=5 THEN//5:00-6:00
JS_ton1[5].IN:=(b_Alarm[4] AND NOT JS_ton1[5].Q);
 
IF JS_ton1[5].Q THEN
	Alarm_CS[5]:=Alarm_CS[5]+1;
END_IF
JS_ton2[5].IN:=(P3_SystemRUN.iMode=1 AND NOT JS_ton2[5].Q );

IF JS_ton2[5].Q THEN
	Auto_CS[5]:=Auto_CS[5]+1;
	
END_IF

Manul_CS[5]:=3600-(Alarm_CS[5]+Auto_CS[5]);

END_IF


JS_ton1[6](PT:=T#1000MS);
JS_ton2[6](PT:=T#1000MS);
IF HMI_Hour=6 THEN//6:00-7:00
JS_ton1[6].IN:=(b_Alarm[4] AND NOT JS_ton1[6].Q);
 
IF JS_ton1[6].Q THEN
	Alarm_CS[6]:=Alarm_CS[6]+1;
END_IF
JS_ton2[6].IN:=(P3_SystemRUN.iMode=1 AND NOT JS_ton2[6].Q );

IF JS_ton2[6].Q THEN
	Auto_CS[6]:=Auto_CS[6]+1;
	
END_IF

Manul_CS[6]:=3600-(Alarm_CS[6]+Auto_CS[6]);

END_IF



JS_ton1[7](PT:=T#1000MS);
JS_ton2[7](PT:=T#1000MS);
IF HMI_Hour=7 THEN//7:00-8:00
JS_ton1[7].IN:=(b_Alarm[4] AND NOT JS_ton1[7].Q);
 
IF JS_ton1[7].Q THEN
	Alarm_CS[7]:=Alarm_CS[7]+1;
END_IF
JS_ton2[7].IN:=(P3_SystemRUN.iMode=1 AND NOT JS_ton2[7].Q );

IF JS_ton2[7].Q THEN
	Auto_CS[7]:=Auto_CS[7]+1;
	
END_IF

Manul_CS[7]:=3600-(Alarm_CS[7]+Auto_CS[7]);

END_IF


JS_ton1[8](PT:=T#1000MS);
JS_ton2[8](PT:=T#1000MS);
IF HMI_Hour=8 THEN//8:00-9:00
JS_ton1[8].IN:=(b_Alarm[4] AND NOT JS_ton1[8].Q);
 
IF JS_ton1[8].Q THEN
	Alarm_CS[8]:=Alarm_CS[8]+1;
END_IF
JS_ton2[8].IN:=(P3_SystemRUN.iMode=1 AND NOT JS_ton2[8].Q );

IF JS_ton2[8].Q THEN
	Auto_CS[8]:=Auto_CS[8]+1;
	
END_IF

Manul_CS[8]:=3600-(Alarm_CS[8]+Auto_CS[8]);

END_IF



JS_ton1[9](PT:=T#1000MS);
JS_ton2[9](PT:=T#1000MS);
IF HMI_Hour=9 THEN//9:00-10:00
JS_ton1[9].IN:=(b_Alarm[4] AND NOT JS_ton1[9].Q);
 
IF JS_ton1[9].Q THEN
	Alarm_CS[9]:=Alarm_CS[9]+1;
END_IF
JS_ton2[9].IN:=(P3_SystemRUN.iMode=1 AND NOT JS_ton2[9].Q );

IF JS_ton2[9].Q THEN
	Auto_CS[9]:=Auto_CS[9]+1;
	
END_IF

Manul_CS[9]:=3600-(Alarm_CS[9]+Auto_CS[9]);

END_IF


JS_ton1[10](PT:=T#1000MS);
JS_ton2[10](PT:=T#1000MS);
IF HMI_Hour=10 THEN//10:00-11:00
JS_ton1[10].IN:=(b_Alarm[4] AND NOT JS_ton1[10].Q);
 
IF JS_ton1[10].Q THEN
	Alarm_CS[10]:=Alarm_CS[10]+1;
END_IF
JS_ton2[10].IN:=(P3_SystemRUN.iMode=1 AND NOT JS_ton2[10].Q );

IF JS_ton2[10].Q THEN
	Auto_CS[10]:=Auto_CS[10]+1;
	
END_IF

Manul_CS[10]:=3600-(Alarm_CS[10]+Auto_CS[10]);

END_IF


JS_ton1[11](PT:=T#1000MS);
JS_ton2[11](PT:=T#1000MS);
IF HMI_Hour=11 THEN//11:00-12:00
JS_ton1[11].IN:=(b_Alarm[4] AND NOT JS_ton1[11].Q);
 
IF JS_ton1[11].Q THEN
	Alarm_CS[11]:=Alarm_CS[11]+1;
END_IF
JS_ton2[11].IN:=(P3_SystemRUN.iMode=1 AND NOT JS_ton2[11].Q );

IF JS_ton2[11].Q THEN
	Auto_CS[11]:=Auto_CS[11]+1;
	
END_IF

Manul_CS[11]:=3600-(Alarm_CS[11]+Auto_CS[11]);

END_IF



JS_ton1[12](PT:=T#1000MS);
JS_ton2[12](PT:=T#1000MS);
IF HMI_Hour=12 THEN//12:00-13:00
JS_ton1[12].IN:=(b_Alarm[4] AND NOT JS_ton1[12].Q);
 
IF JS_ton1[12].Q THEN
	Alarm_CS[12]:=Alarm_CS[12]+1;
END_IF
JS_ton2[12].IN:=(P3_SystemRUN.iMode=1 AND NOT JS_ton2[12].Q );

IF JS_ton2[12].Q THEN
	Auto_CS[12]:=Auto_CS[12]+1;
	
END_IF

Manul_CS[12]:=3600-(Alarm_CS[12]+Auto_CS[12]);

END_IF


JS_ton1[13](PT:=T#1000MS);
JS_ton2[13](PT:=T#1000MS);
IF HMI_Hour=13 THEN//13:00-14:00
JS_ton1[13].IN:=(b_Alarm[4] AND NOT JS_ton1[13].Q);
 
IF JS_ton1[13].Q THEN
	Alarm_CS[13]:=Alarm_CS[13]+1;
END_IF
JS_ton2[13].IN:=(P3_SystemRUN.iMode=1 AND NOT JS_ton2[13].Q );

IF JS_ton2[13].Q THEN
	Auto_CS[13]:=Auto_CS[13]+1;
	
END_IF

Manul_CS[13]:=3600-(Alarm_CS[13]+Auto_CS[13]);

END_IF



JS_ton1[14](PT:=T#1000MS);
JS_ton2[14](PT:=T#1000MS);
IF HMI_Hour=14 THEN//14:00-15:00
JS_ton1[14].IN:=(b_Alarm[4] AND NOT JS_ton1[14].Q);
 
IF JS_ton1[14].Q THEN
	Alarm_CS[14]:=Alarm_CS[14]+1;
END_IF
JS_ton2[14].IN:=(P3_SystemRUN.iMode=1 AND NOT JS_ton2[14].Q );

IF JS_ton2[14].Q THEN
	Auto_CS[14]:=Auto_CS[14]+1;
	
END_IF

Manul_CS[14]:=3600-(Alarm_CS[14]+Auto_CS[14]);

END_IF


JS_ton1[15](PT:=T#1000MS);
JS_ton2[15](PT:=T#1000MS);
IF HMI_Hour=15 THEN//15:00-16:00
JS_ton1[15].IN:=(b_Alarm[4] AND NOT JS_ton1[15].Q);
 
IF JS_ton1[15].Q THEN
	Alarm_CS[15]:=Alarm_CS[15]+1;
END_IF
JS_ton2[15].IN:=(P3_SystemRUN.iMode=1 AND NOT JS_ton2[15].Q );

IF JS_ton2[15].Q THEN
	Auto_CS[15]:=Auto_CS[15]+1;
	
END_IF

Manul_CS[15]:=3600-(Alarm_CS[15]+Auto_CS[15]);

END_IF


JS_ton1[16](PT:=T#1000MS);
JS_ton2[16](PT:=T#1000MS);
IF HMI_Hour=16 THEN//16:00-17:00
JS_ton1[16].IN:=(b_Alarm[4] AND NOT JS_ton1[16].Q);
 
IF JS_ton1[16].Q THEN
	Alarm_CS[16]:=Alarm_CS[16]+1;
END_IF
JS_ton2[16].IN:=(P3_SystemRUN.iMode=1 AND NOT JS_ton2[16].Q );

IF JS_ton2[16].Q THEN
	Auto_CS[16]:=Auto_CS[16]+1;
	
END_IF

Manul_CS[16]:=3600-(Alarm_CS[16]+Auto_CS[16]);

END_IF


JS_ton1[17](PT:=T#1000MS);
JS_ton2[17](PT:=T#1000MS);
IF HMI_Hour=17 THEN//17:00-18:00
JS_ton1[17].IN:=(b_Alarm[4] AND NOT JS_ton1[17].Q);
 
IF JS_ton1[17].Q THEN
	Alarm_CS[17]:=Alarm_CS[17]+1;
END_IF
JS_ton2[17].IN:=(P3_SystemRUN.iMode=1 AND NOT JS_ton2[17].Q );

IF JS_ton2[17].Q THEN
	Auto_CS[17]:=Auto_CS[17]+1;
	
END_IF

Manul_CS[17]:=3600-(Alarm_CS[17]+Auto_CS[17]);

END_IF


JS_ton1[18](PT:=T#1000MS);
JS_ton2[18](PT:=T#1000MS);
IF HMI_Hour=18 THEN//18:00-19:00
JS_ton1[18].IN:=(b_Alarm[4] AND NOT JS_ton1[18].Q);
 
IF JS_ton1[18].Q THEN
	Alarm_CS[18]:=Alarm_CS[18]+1;
END_IF
JS_ton2[18].IN:=(P3_SystemRUN.iMode=1 AND NOT JS_ton2[18].Q );

IF JS_ton2[18].Q THEN
	Auto_CS[18]:=Auto_CS[18]+1;
	
END_IF

Manul_CS[18]:=3600-(Alarm_CS[18]+Auto_CS[18]);

END_IF


JS_ton1[19](PT:=T#1000MS);
JS_ton2[19](PT:=T#1000MS);
IF HMI_Hour=19 THEN//19:00-20:00
JS_ton1[19].IN:=(b_Alarm[4] AND NOT JS_ton1[19].Q);
 
IF JS_ton1[19].Q THEN
	Alarm_CS[19]:=Alarm_CS[19]+1;
END_IF
JS_ton2[19].IN:=(P3_SystemRUN.iMode=1 AND NOT JS_ton2[19].Q );

IF JS_ton2[19].Q THEN
	Auto_CS[19]:=Auto_CS[19]+1;
	
END_IF

Manul_CS[19]:=3600-(Alarm_CS[19]+Auto_CS[19]);

END_IF


JS_ton1[20](PT:=T#1000MS);
JS_ton2[20](PT:=T#1000MS);
IF HMI_Hour=20 THEN//20:00-21:00
JS_ton1[20].IN:=(b_Alarm[4] AND NOT JS_ton1[20].Q);
 
IF JS_ton1[20].Q THEN
	Alarm_CS[20]:=Alarm_CS[20]+1;
END_IF
JS_ton2[20].IN:=(P3_SystemRUN.iMode=1 AND NOT JS_ton2[20].Q );

IF JS_ton2[20].Q THEN
	Auto_CS[20]:=Auto_CS[20]+1;
	
END_IF

Manul_CS[20]:=3600-(Alarm_CS[20]+Auto_CS[20]);

END_IF


JS_ton1[21](PT:=T#1000MS);
JS_ton2[21](PT:=T#1000MS);
IF HMI_Hour=21 THEN//21:00-22:00
JS_ton1[21].IN:=(b_Alarm[4] AND NOT JS_ton1[21].Q);
 
IF JS_ton1[21].Q THEN
	Alarm_CS[21]:=Alarm_CS[21]+1;
END_IF
JS_ton2[21].IN:=(P3_SystemRUN.iMode=1 AND NOT JS_ton2[21].Q );

IF JS_ton2[21].Q THEN
	Auto_CS[21]:=Auto_CS[21]+1;
	
END_IF

Manul_CS[21]:=3600-(Alarm_CS[21]+Auto_CS[21]);

END_IF


JS_ton1[22](PT:=T#1000MS);
JS_ton2[22](PT:=T#1000MS);
IF HMI_Hour=22 THEN//22:00-23:00
JS_ton1[22].IN:=(b_Alarm[4] AND NOT JS_ton1[22].Q);
 
IF JS_ton1[22].Q THEN
	Alarm_CS[22]:=Alarm_CS[22]+1;
END_IF
JS_ton2[22].IN:=(P3_SystemRUN.iMode=1 AND NOT JS_ton2[22].Q );

IF JS_ton2[22].Q THEN
	Auto_CS[22]:=Auto_CS[22]+1;
	
END_IF

Manul_CS[22]:=3600-(Alarm_CS[22]+Auto_CS[22]);

END_IF


JS_ton1[23](PT:=T#1000MS);
JS_ton2[23](PT:=T#1000MS);
IF HMI_Hour=23 THEN//23:00-00:00
JS_ton1[23].IN:=(b_Alarm[4] AND NOT JS_ton1[23].Q);
 
IF JS_ton1[23].Q THEN
	Alarm_CS[23]:=Alarm_CS[23]+1;
END_IF
JS_ton2[23].IN:=(P3_SystemRUN.iMode=1 AND NOT JS_ton2[23].Q );

IF JS_ton2[23].Q THEN
	Auto_CS[23]:=Auto_CS[23]+1;
	
END_IF

Manul_CS[23]:=3600-(Alarm_CS[23]+Auto_CS[23]);

END_IF


//DayClear(CLK:=(HMI_Hour=8 AND HMI_Minute=0 AND HMI_Second=0 ) , Q=> );
//NightClear(CLK:=(HMI_Hour=20 AND HMI_Minute=0 AND HMI_Second=0) , Q=> );



IF Day_Clear OR  DayClear.Q  THEN
	Auto_CS[8]:=0;
	Auto_CS[9]:=0;
	Auto_CS[10]:=0;
	Auto_CS[11]:=0;
	Auto_CS[12]:=0;
	Auto_CS[13]:=0;
	Auto_CS[14]:=0;
	Auto_CS[15]:=0;
	Auto_CS[16]:=0;
	Auto_CS[17]:=0;
	Auto_CS[18]:=0;
	Auto_CS[19]:=0;
	
	Alarm_CS[8]:=0;
	Alarm_CS[9]:=0;
	Alarm_CS[10]:=0;
	Alarm_CS[11]:=0;
	Alarm_CS[12]:=0;
	Alarm_CS[13]:=0;
	Alarm_CS[14]:=0;
	Alarm_CS[15]:=0;
	Alarm_CS[16]:=0;
	Alarm_CS[17]:=0;
	Alarm_CS[18]:=0;
	Alarm_CS[19]:=0;
	
	Manul_CS[8]:=0;
	Manul_CS[9]:=0;
	Manul_CS[10]:=0;
	Manul_CS[11]:=0;
	Manul_CS[12]:=0;
	Manul_CS[13]:=0;
	Manul_CS[14]:=0;
	Manul_CS[15]:=0;
	Manul_CS[16]:=0;
	Manul_CS[17]:=0;
	Manul_CS[18]:=0;
	Manul_CS[19]:=0;
	
END_IF

IF Night_Clear OR NightClear.Q THEN
	Auto_CS[0]:=0;
	Auto_CS[1]:=0;
	Auto_CS[2]:=0;
	Auto_CS[3]:=0;
	Auto_CS[4]:=0;
	Auto_CS[5]:=0;
	Auto_CS[6]:=0;
	Auto_CS[7]:=0;
	Auto_CS[20]:=0;
	Auto_CS[21]:=0;
	Auto_CS[22]:=0;
	Auto_CS[23]:=0;
	
	Alarm_CS[0]:=0;
	Alarm_CS[1]:=0;
	Alarm_CS[2]:=0;
	Alarm_CS[3]:=0;
	Alarm_CS[4]:=0;
	Alarm_CS[5]:=0;
	Alarm_CS[6]:=0;
	Alarm_CS[7]:=0;
	Alarm_CS[20]:=0;
	Alarm_CS[21]:=0;
	Alarm_CS[22]:=0;
	Alarm_CS[23]:=0;
	
	Manul_CS[0]:=0;
	Manul_CS[1]:=0;
	Manul_CS[2]:=0;
	Manul_CS[3]:=0;
	Manul_CS[4]:=0;
	Manul_CS[5]:=0;
	Manul_CS[6]:=0;
	Manul_CS[7]:=0;
	Manul_CS[20]:=0;
	Manul_CS[21]:=0;
	Manul_CS[22]:=0;
	Manul_CS[23]:=0;	

	
END_IF



//运行时间统计
P3TimeData(
	Alm:= b_Alarm[4] , 
	Wait:=P3_SystemRUN.iMode=3 AND NOT b_Alarm[4] , 
	Run:=P3_SystemRUN.iMode=1 , 
	XL_Wait:=(Step36=1910 OR Step36=1917 ) AND P3_SystemRUN.iMode=1  , 
	Query:=HDQuery, 
	date1:=HDdate , 	
	STTimedata=> );

//稼动率
OEE1(
	Alm:=M_Sys .p1state=4 OR  M_Sys .p1state=5 OR 
               P2M1_DTSysState.bErrorStop OR  P2M1_WJSysState.bErrorStop OR
               P2M2_DTSysState.bErrorStop OR  P2M2_WJSysState.bErrorStop OR
               P2M3_DTSysState.bErrorStop OR  P2M3_WJSysState.bErrorStop OR
               b_Alarm[4]  , 
	Wait:= , 
	Run:=  M_Sys .p1state=1 AND
                 P2M1_MachCtrl.U.DT_iMode=1 AND P2M1_MachCtrl.U.WJ_iMode=1 AND P2M1_MachCtrl.U.TJ_iMode=1 AND 
                 P2M2_MachCtrl.U.DT_iMode=1 AND P2M2_MachCtrl.U.WJ_iMode=1 AND P2M2_MachCtrl.U.TJ_iMode=1  AND
                 P2M3_MachCtrl.U.DT_iMode=1 AND P2M3_MachCtrl.U.WJ_iMode=1 AND P2M3_MachCtrl.U.TJ_iMode=1   AND
                 P3_SystemRUN.iMode=1, 
	OEE=> OEE );
*)

END_PROGRAM

// ---- P3POUs/P3FB/FB_ProductionDataLocal.TcPOU
FUNCTION_BLOCK FB_ProductionDataLocal

VAR_INPUT
	NowTimeData	:TIMESTRUCT;(*当前系统时间*)
	OutFlag1:BOOL;(*产量计数标志1*)
	OutFlag2:BOOL;(*产量计数标志2*)
	NGFlag:ARRAY[1..30] OF BOOL;(*NG计数标志*)

	RunFlag:BOOL;(*运行标志*)
	WaitFlag:BOOL;(*待料标志*)
	AlarmFlag:BOOL;(*故障标志*)
	DelDataAMBtn:BOOL;(*白班数据清除按钮*)
	DelDataPMBtn:BOOL;(*夜班数据清除按钮*)
	NGClearAMBtn:ARRAY[1..30] OF BOOL;//白班NG类型计数清零
	NGClearPMBtn:ARRAY[1..30] OF BOOL;//夜班NG类型计数清零
END_VAR



VAR_OUTPUT
	NowOutTotal:REAL;(*当前班次加工总数*)
	NowRate:REAL;(*当前班次良率*)
	OEE:REAL;//稼动率
END_VAR

VAR_IN_OUT
	NowDay				:INT;(*数据移位时所保存当前日*)
	NowMonth			:INT;(*数据移位时所保存当前月*)
	DayHistory			:ARRAY[1..7 ] 	OF INT;(*历史日*)
	MonthHistory		:ARRAY[1..7 ] 	OF INT;(*历史月*)
	TodayTotal:REAL;(*当天24H生产总数*)
	TodayOK:REAL;(*当天24H生产OK总数*)
	TodayNG:REAL;(*当天24H生产NG总数*)
	TodayTotal_AM:REAL;(*当天白班生产总数*)
	TodayTotal_PM:REAL;(*当天夜班生产总数*)
	TodayRate_AM:REAL;(*当天白班良率*)
	TodayRate_PM:REAL;(*当天夜班良率*)
	TodayOK_AM:REAL;(*当天白班生产OK总数*)
	TodayOK_PM:REAL;(*当天夜班生产OK总数*)
	TodayNG_AM:REAL;(*当天白班生产NG总数*)
	TodayNG_PM:REAL;(*当天夜班生产NG总数*)
	TodayHour_AM		:ARRAY[8..19 ] 	OF REAL;(*当天白班每小时产量ARRAY[8..19 ]*)
	TodayHour_PM		:ARRAY[0..23] 	OF REAL;(*当天夜班每小时产量ARRAY[0..23]*)
	TodayNGClass_AM		:ARRAY[1..30 ] 	OF REAL;(*当天白班各类NG数量ARRAY[1..30 ]*)
	TodayNGClass_PM		:ARRAY[1..30 ] 	OF REAL;(*当天夜班各类NG数量ARRAY[1..30 ]*)
	TodayRun_AM			:REAL;(*当天白班总运行时间合计/分*)
	TodayRun_PM			:REAL;(*当天夜班总运行时间合计/分*)
	TodayWait_AM		:REAL;(*当天白班总待料时间合计/分*)
	TodayWait_PM		:REAL;(*当天夜班总待料时间合计/分*)
	TodayAlarm_AM		:REAL;(*当天白班总报警时间合计/分*)
	TodayAlarm_PM		:REAL;(*当天夜班总报警时间合计/分*)

	RunCnt_AM:ARRAY[8..19 ] 	OF UDINT;	(*白班运行时间计数*)
	RunCnt_PM:ARRAY[0..23] 		OF UDINT;	(*夜班运行时间计数*)
	WaitCnt_AM:ARRAY[8..19 ] 	OF UDINT;	(*白班待料时间计数*)
	WaitCnt_PM:ARRAY[0..23] 	OF UDINT;	(*夜班待料时间计数*)
	AlarmCnt_AM:ARRAY[8..19 ] 	OF UDINT;	(*白班报警时间计数*)
	AlarmCnt_PM:ARRAY[0..23] 	OF UDINT;	(*夜班报警时间计数*)

	TodayRun_AMH:ARRAY[8..19 ] OF REAL;(*当天白班每小时运行时间合计/分*)
	TodayRun_PMH:ARRAY[0..23]OF REAL;(*当天夜班每小时运行时间合计/分*)
	TodayWait_AMH:ARRAY[8..19 ] OF REAL;(*当天白班每小时待料时间合计/分*)
	TodayWait_PMH:ARRAY[0..23]OF REAL;(*当天夜班每小时待料时间合计/分*)
	TodayAlarm_AMH	:ARRAY[8..19 ] 	OF	REAL;(*当天白班每小时报警时间合计/分*)
	TodayAlarm_PMH	:ARRAY[0..23]OF REAL;(*当天夜班每小时报警时间合计/分*)

	HistoryTotal:ARRAY[1..7 ] OF REAL;(*历史每天24H生产总数ARRAY[1..7 ]*)
	HistoryOK:ARRAY[1..7 ] OF REAL;(*历史每天24H生产OK总数ARRAY[1..7 ]*)
	HistoryNG:ARRAY[1..7 ] OF REAL;(*历史每天24H生产NG总数ARRAY[1..7 ]*)
	HistoryTotal_AM:ARRAY[1..7 ] OF REAL;(*历史每天白班生产总数ARRAY[1..7 ]*)
	HistoryTotal_PM:ARRAY[1..7 ] OF REAL;(*历史每天夜班生产总数ARRAY[1..7 ]*)
	HistoryRate_AM:ARRAY[1..7 ] OF REAL;(*历史每天白班良率ARRAY[1..7 ]*)
	HistoryRate_PM:ARRAY[1..7 ] OF REAL;(*历史每天夜班良率ARRAY[1..7 ]*)
	HistoryOK_AM:ARRAY[1..7 ] OF REAL;(*历史每天白班生产OK总数ARRAY[1..7 ]*)
	HistoryOK_PM:ARRAY[1..7 ] OF REAL;(*历史每天夜班生产OK总数ARRAY[1..7 ]*)
	HistoryNG_AM:ARRAY[1..7 ] OF REAL;(*历史每天白班生产NG总数ARRAY[1..7 ]*)
	HistoryNG_PM:ARRAY[1..7 ] OF REAL;(*历史每天夜班生产NG总数ARRAY[1..7 ]*)
	HistoryHour_AM		:ARRAY[1..7,8..19 ] 	OF REAL;(*历史每天白班每小时产量ARRAY[1..7,8..19 ]*)
	HistoryHour_PM		:ARRAY[1..7,0..23] 		OF REAL;(*历史每天夜班每小时产量ARRAY[1..7,0..23]*)
	HistoryNGClass_AM	:ARRAY[1..7,1..30 ] 	OF REAL;(*历史每天白班各类NG数量ARRAY[1..7,1..30 ]*)
	HistoryNGClass_PM	:ARRAY[1..7,1..30 ] 	OF REAL;(*历史每天夜班各类NG数量ARRAY[1..7,1..30 ]*)
	HistoryRun_AM		:ARRAY[1..7 ] OF REAL;(*历史每天白班总运行时间合计ARRAY[1..7 ]*)
	HistoryRun_PM		:ARRAY[1..7 ] OF REAL;(*历史每天夜班总运行时间合计ARRAY[1..7 ]*)
	HistoryWait_AM		:ARRAY[1..7 ] OF REAL;(*历史每天白班总待料时间合计ARRAY[1..7 ]*)
	HistoryWait_PM		:ARRAY[1..7 ] OF REAL;(*历史每天夜班总待料时间合计ARRAY[1..7 ]*)
	HistoryAlarm_AM		:ARRAY[1..7 ] OF REAL;(*历史每天白班总报警时间合计ARRAY[1..7 ]*)
	HistoryAlarm_PM		:ARRAY[1..7 ] OF REAL;(*历史每天夜班总报警时间合计ARRAY[1..7 ]*)

	HistoryRun_AMH		:ARRAY[1..7,8..19 ] OF REAL;(*历史每天白班每小时运行时间合计ARRAY[1..7 ]*)
	HistoryRun_PMH		:ARRAY[1..7,0..23 ] OF REAL;(*历史每天夜班每小时运行时间合计ARRAY[1..7 ]*)
	HistoryWait_AMH		:ARRAY[1..7,8..19 ] OF REAL;(*历史每天白班每小时待料时间合计ARRAY[1..7 ]*)
	HistoryWait_PMH		:ARRAY[1..7,0..23 ] OF REAL;(*历史每天夜班每小时待料时间合计ARRAY[1..7 ]*)
	HistoryAlarm_AMH	:ARRAY[1..7,8..19 ] OF REAL;(*历史每天白班每小时报警时间合计ARRAY[1..7 ]*)
	HistoryAlarm_PMH	:ARRAY[1..7,0..23 ] OF REAL;(*历史每天夜班每小时报警时间合计ARRAY[1..7 ]*)
	
	TodayNgHour_Day:ARRAY[1..30,0..23] OF REAL;//白班每小时NG类型统计,,
	TodayNgHour_Night:ARRAY[1..30,0..23] OF REAL;//夜班每小时NG类型统计,,
	HisTodayNgHour_Day:ARRAY[1..30,0..23,1..7] OF REAL;//l历史白班每小时NG类型统计,,
	HisTodayNgHour_Night:ARRAY[1..30,0..23,1..7] OF REAL;//历史夜班每小时NG类型统计,,
END_VAR


VAR
	i:INT;
	j: INT;
	K:INT;
	m:INT;
	TrigOutAdd1:R_TRIG ;	(*产量计数上升沿1*)
	TrigOutAdd2:R_TRIG ;	(*产量计数上升沿1*)
	TrigNgAdd: ARRAY[1..30 ] OF R_TRIG;(*1-30类ng计数统计*)
	HistoryData_Step:UINT;(*历史数据保存步*)
	SaveDataDelay:TON;(*历史数据保存延时，防止处理周期内多次存储*)
	rNGClearAMBtn:ARRAY [1..30] OF R_TRIG;//白班ng类型清零上升沿
	rNGClearPMBtn:ARRAY [1..30] OF R_TRIG;//夜班NG类型清零上升沿
	
	

END_VAR


(**********************  分段产能  ***************************************)
TrigOutAdd1(CLK:=OutFlag1,Q=> );(*产量计数上升沿1*)
TrigOutAdd2(CLK:=OutFlag2,Q=> );(*产量计数上升沿1*)
FOR i:=1 TO 30 DO
	rNGClearAMBtn[i](CLK:=NGClearAMBtn[i],Q=> );//白班ng类型清零上升沿
	rNGClearPMBtn[i](CLK:=NGClearPMBtn[i],Q=> );//夜班NG类型清零上升沿
END_FOR
FOR m:=1 TO 30 DO
	IF  rNGClearAMBtn[m].Q THEN
		TodayNGClass_AM[m]:=0;
	END_IF
	IF  rNGClearPMBtn[m].Q THEN
		TodayNGClass_PM[m]:=0;
	END_IF
END_FOR
//NG分类统计触发
TrigNgAdd[1](CLK:=NGFlag[1],Q=> );(*1类ng*)//扫码NG
TrigNgAdd[2](CLK:=NGFlag[2],Q=> );(*2类ng*)//短路测试NG
TrigNgAdd[3](CLK:=NGFlag[3],Q=> );(*3类ng*)//称重NG
TrigNgAdd[4](CLK:=NGFlag[4],Q=> );(*4类ng*)//测厚NG
TrigNgAdd[5](CLK:=NGFlag[5],Q=> );(*5类ng*)//MES卡站不良
TrigNgAdd[6](CLK:=NGFlag[6],Q=> );(*6类ng*)//烤箱超时NG
TrigNgAdd[7](CLK:=NGFlag[7],Q=> );(*7类ng*)//1号叠台对齐度NG数
TrigNgAdd[8](CLK:=NGFlag[8],Q=> );(*8类ng*)//2号叠台对齐度NG数
TrigNgAdd[9](CLK:=NGFlag[9],Q=> );(*9类ng*)//3号叠台对齐度NG数
TrigNgAdd[10](CLK:=NGFlag[10],Q=> );(*10类ng*)//1号叠台首检NG数
TrigNgAdd[11](CLK:=NGFlag[11],Q=> );(*11类ng*)//2号叠台首检NG数
TrigNgAdd[12](CLK:=NGFlag[12],Q=> );(*12类ng*)//3号叠台首检NG数
TrigNgAdd[13](CLK:=NGFlag[13],Q=> );(*13类ng*)//模切正极NG数
TrigNgAdd[14](CLK:=NGFlag[14],Q=> );(*14类ng*)//模切负极NG数
TrigNgAdd[15](CLK:=NGFlag[15],Q=> );(*15类ng*)//正极纠偏平台NG数
TrigNgAdd[16](CLK:=NGFlag[16],Q=> );(*16类ng*)//负极纠偏平台NG数
TrigNgAdd[17](CLK:=NGFlag[17],Q=> );(*17类ng*)//正极对齐度NG数
TrigNgAdd[18](CLK:=NGFlag[18],Q=> );(*18类ng*)//负极对齐度NG数
TrigNgAdd[19](CLK:=NGFlag[19],Q=> );(*19类ng*)
TrigNgAdd[20](CLK:=NGFlag[20],Q=> );(*20类ng*)
TrigNgAdd[21](CLK:=NGFlag[21],Q=> );(*21类ng*)
TrigNgAdd[22](CLK:=NGFlag[22],Q=> );(*22类ng*)
TrigNgAdd[23](CLK:=NGFlag[23],Q=> );(*23类ng*)
TrigNgAdd[24](CLK:=NGFlag[24],Q=> );(*24类ng*)
TrigNgAdd[25](CLK:=NGFlag[25],Q=> );(*25类ng*)
TrigNgAdd[26](CLK:=NGFlag[26],Q=> );(*26类ng*)
TrigNgAdd[27](CLK:=NGFlag[27],Q=> );(*27类ng*)
TrigNgAdd[28](CLK:=NGFlag[28],Q=> );(*28类ng*)
TrigNgAdd[29](CLK:=NGFlag[29],Q=> );(*29类ng*)
TrigNgAdd[30](CLK:=NGFlag[30],Q=> );(*30类ng*)

(***白班数据统计******)
FOR i:=8 TO 19 DO
	IF NowTimeData.wHour=i THEN
		IF i>=8 AND i<=19 THEN
			(********产量计数**********)
			IF TrigOutAdd1.Q  THEN
				TodayHour_AM[i]:=TodayHour_AM[i]+1;
			END_IF
			IF TrigOutAdd2.Q  THEN
				TodayHour_AM[i]:=TodayHour_AM[i]+1;
			END_IF
			(*******白班NG不良分类统计*)
			FOR m:=1 TO 10 DO
				IF TrigNgAdd[m].Q THEN
					TodayNGClass_AM[m]:=TodayNGClass_AM[m]+1;
				END_IF
			END_FOR
			
			(******************白班每小时NG类型统计*******************)
			FOR m:=11 TO 30 DO
					IF TrigNgAdd[m].Q THEN
							TodayNgHour_Day[m,i]:=TodayNgHour_Day[m,i]+1;//白班每小时NG类型统计
					END_IF
			END_FOR
				
				
			 (*运行时间统计*)
			IF RunFlag THEN
				RunCnt_AM[i]:=RunCnt_AM[i]+1;
			END_IF
			TodayRun_AMH[i]:=UDINT_TO_REAL(RunCnt_AM[i]/(500*60)) ;
			 (*待料时间统计*)
			IF  WaitFlag  THEN
				WaitCnt_AM[i]:=WaitCnt_AM[i]+1;
			END_IF
			TodayWait_AMH[i]:=UDINT_TO_REAL(WaitCnt_AM[i]/(500*60)) ;
			(*报警时间统计*)
			IF  AlarmFlag THEN
				AlarmCnt_AM[i]:=AlarmCnt_AM[i]+1;
			END_IF
			TodayAlarm_AMH[i]:=UDINT_TO_REAL(AlarmCnt_AM[i]/(500*60)) ;

			(*当前生产输出*)
			NowOutTotal:=TodayTotal_AM;
			NowRate:=TodayRate_AM;
			
		END_IF
	END_IF
END_FOR

(***手动清除白班产量统计数据******)
IF DelDataAMBtn THEN
	FOR j := 8 TO 19 DO
		TodayHour_AM[j]:=0 ;
		RunCnt_AM[j]:= 0 ;(*白班运行时间计数*)
		AlarmCnt_AM[j]:= 0 ;(*白班报警时间计数*)
		WaitCnt_AM[j]:= 0 ;(*白班待料时间计数*)
		
		RunCnt_AM[j]:=0;
		TodayRun_AMH[j]:=0;
		WaitCnt_AM[j]:=0;
		TodayWait_AMH[j]:=0;
		AlarmCnt_AM[j]:=0;
		TodayAlarm_AMH[j]:=0;
	END_FOR
	(*
	FOR j := 1 TO 20 DO
		TodayNGClass_AM[j] := 0 ;
	END_FOR
	*)
	TodayTotal_AM:=0;(*当天白班生产总数*)
	TodayRate_AM:=0;(*当天白班良率*)
	TodayOK_AM:=0;(*当天白班生产OK总数*)
	TodayNG_AM:=0;(*当天白班生产NG总数*)
	
END_IF
(*当天白班生产总数*)
TodayTotal_AM:=TodayHour_AM[8]+TodayHour_AM[9]+TodayHour_AM[10]+TodayHour_AM[11]+TodayHour_AM[12]+TodayHour_AM[13]+
				TodayHour_AM[14]+TodayHour_AM[15]+TodayHour_AM[16]+TodayHour_AM[17]+TodayHour_AM[18]+TodayHour_AM[19]+
                TodayNGClass_AM[13]+TodayNGClass_AM[15]+TodayNGClass_AM[17];
(*当天白班生产NG总数*)
TodayNG_AM:=TodayNGClass_AM[1]+TodayNGClass_AM[2]+TodayNGClass_AM[3]+TodayNGClass_AM[4]+TodayNGClass_AM[5]+
				TodayNGClass_AM[6](*+TodayNGClass_AM[7]+TodayNGClass_AM[8]+TodayNGClass_AM[9]+TodayNGClass_AM[10]*)+
				TodayNGClass_AM[11]+TodayNGClass_AM[12]+TodayNGClass_AM[13]+TodayNGClass_AM[14]+TodayNGClass_AM[15]+
				TodayNGClass_AM[16]+TodayNGClass_AM[17]+TodayNGClass_AM[18]+TodayNGClass_AM[19]+TodayNGClass_AM[20]+
				TodayNGClass_AM[21]+TodayNGClass_AM[22]+TodayNGClass_AM[23]+TodayNGClass_AM[24]+TodayNGClass_AM[25]+
				TodayNGClass_AM[26]+TodayNGClass_AM[27]+TodayNGClass_AM[28]+TodayNGClass_AM[29]+TodayNGClass_AM[30];
(*当天白班生产OK总数*)
TodayOK_AM:=TodayTotal_AM-TodayNG_AM;
(*当天白班良率*)
IF TodayTotal_AM<>0 THEN
	TodayRate_AM:=100*TodayOK_AM/TodayTotal_AM;
END_IF

(*当天白班总运行时间合计/分*)
TodayRun_AM:=TodayRun_AMH[8]+TodayRun_AMH[9]+TodayRun_AMH[10]+TodayRun_AMH[11]+TodayRun_AMH[12]+TodayRun_AMH[13]+
				TodayRun_AMH[14]+TodayRun_AMH[15]+TodayRun_AMH[16]+TodayRun_AMH[17]+TodayRun_AMH[18]+TodayRun_AMH[19];
(*当天白班总待料时间合计/分*)
TodayWait_AM:=TodayWait_AMH[8]+TodayWait_AMH[9]+TodayWait_AMH[10]+TodayWait_AMH[11]+TodayWait_AMH[12]+TodayWait_AMH[13]+
				TodayWait_AMH[14]+TodayWait_AMH[15]+TodayWait_AMH[16]+TodayWait_AMH[17]+TodayWait_AMH[18]+TodayWait_AMH[19];
(*当天白班总报警时间合计/分*)
TodayAlarm_AM:=TodayAlarm_AMH[8]+TodayAlarm_AMH[9]+TodayAlarm_AMH[10]+TodayAlarm_AMH[11]+TodayAlarm_AMH[12]+TodayAlarm_AMH[13]+
				TodayAlarm_AMH[14]+TodayAlarm_AMH[15]+TodayAlarm_AMH[16]+TodayAlarm_AMH[17]+TodayAlarm_AMH[18]+TodayAlarm_AMH[19];
(***白班数据统计******)


(*******夜班数据统计******)
FOR i:=0 TO 23 DO
	IF NowTimeData.wHour=i THEN
		IF i<=7 OR i>=20 THEN
			(********产量计数**********)
			IF TrigOutAdd1.Q  THEN
				TodayHour_PM[i]:=TodayHour_PM[i]+1;
			END_IF
			IF TrigOutAdd2.Q  THEN
				TodayHour_PM[i]:=TodayHour_PM[i]+1;
			END_IF
			(*******夜班NG不良分类统计*)
			FOR m:= 1 TO 10 DO
				IF TrigNgAdd[m].Q THEN
					TodayNGClass_PM[m]:=TodayNGClass_PM[m]+1;		
				END_IF
			END_FOR
			(******************夜班每小时NG类型统计*******************)
			FOR m:= 11 TO 30 DO
					IF TrigNgAdd[m].Q THEN
							TodayNgHour_Night[m,i]:=TodayNgHour_Night[m,i]+1;//夜班每小时NG类型统计
					END_IF
			END_FOR
			
			 (*运行时间统计*)
			IF RunFlag THEN
				RunCnt_PM[i]:=RunCnt_PM[i]+1;
			END_IF
			TodayRun_PMH[i]:=UDINT_TO_REAL(RunCnt_PM[i]/(500*60)) ;
			 (*待料时间统计*)
			IF  WaitFlag  THEN
				WaitCnt_PM[i]:=WaitCnt_PM[i]+1;
			END_IF
			TodayWait_PMH[i]:=UDINT_TO_REAL(WaitCnt_PM[i]/(500*60)) ;
			(*报警时间统计*)
			IF  AlarmFlag THEN
				AlarmCnt_PM[i]:=AlarmCnt_PM[i]+1;
			END_IF
			TodayAlarm_PMH[i]:=UDINT_TO_REAL(AlarmCnt_PM[i]/(500*60)) ;
			(*当前生产输出*)
			NowOutTotal:=TodayTotal_PM;
			NowRate:=TodayRate_PM;
		END_IF
	END_IF
END_FOR

(***手动清除夜班产量统计数据******)
IF DelDataPMBtn THEN
	FOR j:=0 TO 23 DO
		TodayHour_PM[j]:=0 ;
		RunCnt_PM[j]:= 0 ;(*夜班运行时间计数*)
		AlarmCnt_PM[j]:=0;(*夜班报警时间计数*)
		WaitCnt_PM[j]:= 0 ;(*夜班待料时间计数*)
		RunCnt_PM[j]:=0;
		TodayRun_PMH[j]:=0;
		WaitCnt_PM[j]:=0;
		TodayWait_PMH[j]:=0;
		AlarmCnt_PM[j]:=0;
		TodayAlarm_PMH[j]:=0;
(*
	FOR j := 1 TO 20 DO
		TodayNGClass_PM[j] := 0 ;
	END_FOR
*)
	TodayTotal_PM:=0;(*当天夜班生产总数*)
	TodayRate_PM:=0;(*当天夜班良率*)
	TodayOK_PM:=0;(*当天夜班生产OK总数*)
	TodayNG_PM:=0;(*当天夜班生产NG总数*)
	END_FOR
END_IF

(*当天夜班生产总数*)
TodayTotal_PM:=TodayHour_PM[20]+TodayHour_PM[21]+TodayHour_PM[22]+TodayHour_PM[23]+TodayHour_PM[0]+TodayHour_PM[1]+
					TodayHour_PM[2]+TodayHour_PM[3]+TodayHour_PM[4]+TodayHour_PM[5]+TodayHour_PM[6]+TodayHour_PM[7]+
                    TodayNGClass_PM[13]+TodayNGClass_PM[15]+TodayNGClass_PM[17];
(*当天夜班生产NG总数*)
TodayNG_PM:=TodayNGClass_PM[1]+TodayNGClass_PM[2]+TodayNGClass_PM[3]+TodayNGClass_PM[4]+TodayNGClass_PM[5]+
				TodayNGClass_PM[6](*+TodayNGClass_PM[7]+TodayNGClass_PM[8]+TodayNGClass_PM[9]+TodayNGClass_PM[10]*)+
				TodayNGClass_PM[11]+TodayNGClass_PM[12]+TodayNGClass_PM[13]+TodayNGClass_PM[14]+TodayNGClass_PM[15]+
				TodayNGClass_PM[16]+TodayNGClass_PM[17]+TodayNGClass_PM[18]+TodayNGClass_PM[19]+TodayNGClass_PM[20]+
				TodayNGClass_PM[21]+TodayNGClass_PM[22]+TodayNGClass_PM[23]+TodayNGClass_PM[24]+TodayNGClass_PM[25]+
				TodayNGClass_PM[26]+TodayNGClass_PM[27]+TodayNGClass_PM[28]+TodayNGClass_PM[29]+TodayNGClass_PM[30];
(*当天夜班生产OK总数*)
TodayOK_PM:=TodayTotal_PM-TodayNG_PM;
(*当天夜班良率*)
IF TodayTotal_PM<>0 THEN
	TodayRate_PM:=100*TodayOK_PM/TodayTotal_PM;
END_IF
(*当天夜班总运行时间合计/分*)
TodayRun_PM:=TodayRun_PMH[20]+TodayRun_PMH[21]+TodayRun_PMH[22]+TodayRun_PMH[23]+TodayRun_PMH[0]+TodayRun_PMH[1]+
			TodayRun_PMH[2]+TodayRun_PMH[3]+TodayRun_PMH[4]+TodayRun_PMH[5]+TodayRun_PMH[6]+TodayRun_PMH[7];
(*当天夜班总待料时间合计/分*)
TodayWait_PM:=TodayWait_PMH[20]+TodayWait_PMH[21]+TodayWait_PMH[22]+TodayWait_PMH[23]+TodayWait_PMH[0]+TodayWait_PMH[1]+
			TodayWait_PMH[2]+TodayWait_PMH[3]+TodayWait_PMH[4]+TodayWait_PMH[5]+TodayWait_PMH[6]+TodayWait_PMH[7];
(*当天夜班总报警时间合计/分*)
TodayAlarm_PM:=TodayAlarm_PMH[20]+TodayAlarm_PMH[21]+TodayAlarm_PMH[22]+TodayAlarm_PMH[23]+TodayAlarm_PMH[0]+TodayAlarm_PMH[1]+
			TodayAlarm_PMH[2]+TodayAlarm_PMH[3]+TodayAlarm_PMH[4]+TodayAlarm_PMH[5]+TodayAlarm_PMH[6]+TodayAlarm_PMH[7];

(*******夜班数据统计******)


(*******白班+夜班数据汇总******)
TodayTotal:=TodayTotal_AM+TodayTotal_PM;(*当天生产总数*)
TodayNG:=TodayNG_AM+TodayNG_PM;(*当天生产NG总数*)
TodayOK:=TodayTotal-TodayNG;(*当天生产OK总数*)
(*******白班+夜班数据汇总******)


(*************历史数据存储**************)
CASE HistoryData_Step OF
0:
	IF NowTimeData.wHour>=8 AND NowTimeData.wMinute>=00  AND NowTimeData.wSecond>=00 AND NowDay<>NowTimeData.wDay THEN
		HistoryData_Step:=100;(*8点钟机台断电，错过数据移位。重新移位数据*)
	ELSIF NowTimeData.wHour=8 AND NowTimeData.wMinute=00  AND NowTimeData.wSecond=00 AND NowDay=NowTimeData.wDay THEN
		HistoryData_Step:=100;
	END_IF
100:
(**************************************前一天白班夜班的历史数据移位*************************************************)
	FOR  i :=6 TO 1 BY -1 DO
			DayHistory[i+1]:=DayHistory[i] ;(*日*)
			MonthHistory[i+1]:=MonthHistory[i] ;(*月*)
			HistoryTotal[i+1]:=HistoryTotal[i];(*历史每天生产总数*)
			HistoryOK[i+1]:=HistoryOK[i];(*历史每天生产OK总数*)
			HistoryNG[i+1]:=HistoryNG[i];(*历史每天生产NG总数*)
			HistoryTotal_AM[i+1]:=HistoryTotal_AM[i];(*历史每天白班生产总数*)
			HistoryTotal_PM[i+1]:=HistoryTotal_PM[i];(*历史每天夜班生产总数*)
			HistoryRate_AM[i+1]:=HistoryRate_AM[i];(*历史每天白班良率*)
			HistoryRate_PM[i+1]:=HistoryRate_PM[i];(*历史每天夜班良率*)
			HistoryOK_AM[i+1]:=HistoryOK_AM[i];(*历史每天白班生产OK总数*)
			HistoryOK_PM[i+1]:=HistoryOK_PM[i];(*历史每天夜班生产OK总数*)
			HistoryNG_AM[i+1]:=HistoryNG_AM[i];(*历史每天白班生产NG总数*)
			HistoryNG_PM[i+1]:=HistoryNG_PM[i];(*历史每天夜班生产NG总数*)
			HistoryRun_AM[i+1]:=HistoryRun_AM[i];(*历史每天白班总运行时间合计*)
			HistoryRun_PM[i+1]:=HistoryRun_PM[i];(*历史每天夜班总运行时间合计*)
			HistoryWait_AM[i+1]:=HistoryWait_AM[i];(*历史每天白班总待料时间合计*)
			HistoryWait_PM[i+1]:=HistoryWait_PM[i];(*历史每天夜班总待料时间合计*)
			HistoryAlarm_AM[i+1]:=HistoryAlarm_AM[i];(*历史每天白班总报警时间合计*)
			HistoryAlarm_PM[i+1]:=HistoryAlarm_PM[i];(*历史每天夜班总报警时间合计*)

			FOR j := 1 TO 30 DO(*i表示天数，j表示1-10不良分类*)
				HistoryNGClass_AM[i+1,j]:=HistoryNGClass_AM[i,j];(*历史每天白班各类NG数量*)
				HistoryNGClass_PM[i+1,j]:=HistoryNGClass_PM[i,j];(*历史每天夜班各类NG数量*)
			END_FOR
			FOR j := 8 TO 19 DO(*j表示小时*)
				HistoryHour_AM[i+1,j]:=HistoryHour_AM[i,j];(*历史每天白班每小时产量*)
				HistoryRun_AMH[i+1,j]:=HistoryRun_AMH[i,j];(*历史每天白班每小时运行时间合计ARRAY[1..7 ]*)
				HistoryWait_AMH[i+1,j]:=HistoryWait_AMH[i,j];(*历史每天白班每小时待料时间合计ARRAY[1..7 ]*)
				HistoryAlarm_AMH[i+1,j]:=HistoryAlarm_AMH[i,j];(*历史每天白班每小时报警时间合计ARRAY[1..7 ]*)
			END_FOR
			FOR j := 0 TO 23 DO(*j表示小时*)
				HistoryHour_PM[i+1,j]:=HistoryHour_PM [i,j];(*夜班移位每小时产量*)
				HistoryRun_PMH[i+1,j]:=HistoryRun_PMH[i,j];(*历史每天夜班每小时运行时间合计ARRAY[1..7 ]*)
				HistoryWait_PMH[i+1,j]:=HistoryWait_PMH[i,j];(*历史每天夜班每小时待料时间合计ARRAY[1..7 ]*)
				HistoryAlarm_PMH[i+1,j]:=HistoryAlarm_PMH[i,j];(*历史每天夜班每小时报警时间合计ARRAY[1..7 ]*)
			END_FOR
			FOR j:=0 TO 23 DO//j表示小时
				FOR m:=1 TO 30 DO//m表示多少种NG类型
						HisTodayNgHour_Day[m,j,i+1] :=HisTodayNgHour_Day[m,j,i];//l历史白班每小时NG类型统计,,
						HisTodayNgHour_Night[m,j,i+1]:=HisTodayNgHour_Night[m,j,i];//历史夜班每小时NG类型统计,,
				END_FOR
			END_FOR
	END_FOR
	HistoryData_Step:=200;
200:
(*******将当天日期和数据传送到历史数据存储区***************)
	DayHistory[1]:= NowDay;
	MonthHistory[1]:=NowMonth;
	HistoryTotal[1]:=TodayTotal;(*历史每天生产总数*)
	HistoryOK[1]:=TodayOK;(*历史每天生产OK总数*)
	HistoryNG[1]:=TodayNG;(*历史每天生产NG总数*)
	HistoryTotal_AM[1]:=TodayTotal_AM;(*历史每天白班生产总数*)
	HistoryTotal_PM[1]:=TodayTotal_PM;(*历史每天夜班生产总数*)
	HistoryRate_AM[1]:=TodayRate_AM;(*历史每天白班良率*)
	HistoryRate_PM[1]:=TodayRate_PM;(*历史每天夜班良率*)
	HistoryOK_AM[1]:=TodayOK_AM;(*历史每天白班生产OK总数*)
	HistoryOK_PM[1]:=TodayOK_PM;(*历史每天夜班生产OK总数*)
	HistoryNG_AM[1]:=TodayNG_AM;(*历史每天白班生产NG总数*)
	HistoryNG_PM[1]:=TodayNG_PM;(*历史每天夜班生产NG总数*)
	HistoryRun_AM	[1]:=TodayRun_AM;(*历史每天白班总运行时间合计*)
	HistoryRun_PM[1]:=TodayRun_PM;(*历史每天夜班总运行时间合计*)
	HistoryWait_AM[1]:=TodayWait_AM;(*历史每天白班总待料时间合计*)
	HistoryWait_PM[1]:=TodayWait_PM;(*历史每天夜班总待料时间合计*)
	HistoryAlarm_AM[1]:=TodayAlarm_AM;(*历史每天白班总报警时间合计*)
	HistoryAlarm_PM[1]:=TodayAlarm_PM;(*历史每天夜班总报警时间合计*)
	FOR j := 1 TO 30 DO(*i表示天数，j表示1-30不良分类*)
		HistoryNGClass_AM[1,j]:=TodayNGClass_AM[j];(*历史每天白班各类NG数量*)
		HistoryNGClass_PM[1,j]:=TodayNGClass_PM[j];(*历史每天夜班各类NG数量*)
	END_FOR
	FOR j := 8 TO 19 DO(*j表示小时*)
		HistoryHour_AM[1,j]:=TodayHour_AM[j];(*历史每天白班每小时产量*)
		HistoryRun_AMH[1,j]:=TodayRun_AMH[j];(*历史每天白班每小时运行时间合计ARRAY[1..7 ]*)
		HistoryWait_AMH[1,j]:=TodayWait_AMH[j];(*历史每天白班每小时待料时间合计ARRAY[1..7 ]*)
		HistoryAlarm_AMH[1,j]:=TodayAlarm_AMH[j];(*历史每天白班每小时报警时间合计ARRAY[1..7 ]*)
	END_FOR
	FOR j := 0 TO 23 DO(*j表示小时*)
		HistoryHour_PM[1,j]:=TodayHour_PM [j];(*夜班移位每小时产量*)
		HistoryRun_PMH[1,j]:=TodayRun_PMH[j];(*历史每天夜班每小时运行时间合计ARRAY[1..7 ]*)
		HistoryWait_PMH[1,j]:=TodayWait_PMH[j];(*历史每天夜班每小时待料时间合计ARRAY[1..7 ]*)
		HistoryAlarm_PMH[1,j]:=TodayAlarm_PMH[j];(*历史每天夜班每小时报警时间合计ARRAY[1..7 ]*)
	END_FOR
	
	FOR j:=0 TO 23 DO
		FOR i:=1 TO 30 DO
				HisTodayNgHour_Day[i,j,1] :=TodayNgHour_Day[i,j];//l历史白班每小时NG类型统计,,
				HisTodayNgHour_Night[i,j,1]:=TodayNgHour_Night[i,j];//历史夜班每小时NG类型统计,,
		END_FOR
	END_FOR
	HistoryData_Step:=300;
300:
(******清除当天数据，并记录当天日期*******)
	NowDay:=NowTimeData.wDay;
	NowMonth:=NowTimeData.wMonth;
	FOR i:=8 TO 19 DO
		TodayHour_AM[i]:=0;(*当天白班每小时产量*)
		RunCnt_AM[i]:=0;		(*白班运行时间计数*)
		WaitCnt_AM[i]:=0;	(*白班待料时间计数*)
		AlarmCnt_AM[i]:=0;	(*白班报警时间计数*)
		TodayRun_AMH[i]:=0;
		TodayWait_AMH[i]:=0;
		TodayAlarm_AMH[i]:=0;
	END_FOR
	FOR i:=0 TO 23 DO
		TodayHour_PM[i]:=0;(*当天夜班每小时产量*)
		RunCnt_PM[i]:=0;		(*夜班运行时间计数*)
		WaitCnt_PM[i]:=0;	(*夜班待料时间计数*)
		AlarmCnt_PM[i]:=0;	(*夜班报警时间计数*)
		TodayRun_PMH[i]:=0;
		TodayWait_PMH[i]:=0;
		TodayAlarm_PMH[i]:=0;
	END_FOR
	FOR i:=1 TO 30 DO
		TodayNGClass_AM[i]:=0;(*当天白班各类NG数量*)
		TodayNGClass_PM[i]:=0;(*当天夜班各类NG数量*)
	END_FOR
	TodayTotal:=0;(*当天生产总数*)
	TodayOK:=0;(*当天生产OK总数*)
	TodayNG:=0;(*当天生产NG总数*)
	TodayTotal_AM:=0;(*当天白班生产总数*)
	TodayTotal_PM:=0;(*当天夜班生产总数*)
	TodayRate_AM:=0;(*当天白班良率*)
	TodayRate_PM:=0;(*当天夜班良率*)
	TodayOK_AM:=0;(*当天白班生产OK总数*)
	TodayOK_PM:=0;(*当天夜班生产OK总数*)
	TodayNG_AM:=0;(*当天白班生产NG总数*)
	TodayNG_PM:=0;(*当天夜班生产NG总数*)
	TodayRun_AM:=0;(*当天白班总运行时间合计*)
	TodayRun_PM:=0;(*当天夜班总运行时间合计*)
	TodayWait_AM:=0;(*当天白班总待料时间合计*)
	TodayWait_PM:=0;(*当天夜班总待料时间合计*)
	TodayAlarm_AM:=0;(*当天白班总报警时间合计*)
	TodayAlarm_PM:=0;(*当天夜班总报警时间合计*)	
	FOR i:=1 TO 30 DO
		FOR j:= 0 TO 23 DO
			TodayNgHour_Day[i,j]:=0;//白班每小时NG类型统计,,
			TodayNgHour_Night[i,j]:=0;//夜班每小时NG类型统计,,
		END_FOR
	END_FOR
	SaveDataDelay(IN:=FALSE);
	HistoryData_Step:=400;
400:
	SaveDataDelay(IN:=TRUE,PT:=t#2s, Q=> , ET=> );
	IF SaveDataDelay.Q THEN
		SaveDataDelay(IN:=FALSE);
		HistoryData_Step:=0;
	END_IF
END_CASE
(*************历史数据存储**************)




//	OEE稼动率:=24小时总运行时间/总报警时间+总运行时间
OEE:=(TodayRun_AM+TodayRun_PM)/((TodayRun_AM+TodayRun_PM)+(TodayAlarm_AM+TodayAlarm_PM));

END_FUNCTION_BLOCK

// ---- P3POUs/POUs/Auxiliary/MES_JT_ZT.TcPOU
PROGRAM MES_JT_ZT
VAR
	status_switching:R_TRIG;
    status_switching2:R_TRIG;
	Equipment_parameter_check_R:R_TRIG;
    Bullet_window1 : BOOL ;//弹窗条件
    Bullet_window2 : BOOL ;//弹窗
    Bounce_TON :TON ;//弹窗延时
    Status_switching_TON :TON ;//状态切换延时
    Status_switching2_TON :TON ;//状态切换延时2
    Standby_TON :TON;//待料状态切换延时
	
	ExcelRate_R	:R_TRIG;	//Mes读取优报表
	MTDExcelRate_R:R_TRIG;	//模切给叠台数据完成
	Mes1RdStep	:UINT;	//Mes1读数据步	
	tonWaitMQdata	:TON;	//等待模切数据超时
	ton2	:TON;
	rt:R_TRIG;
END_VAR


status_switching(CLK:=Device_Status_code=9  , Q=> );
status_switching2(CLK:=Device_Status_code=18  , Q=> ); 
IF status_switching.Q OR status_switching2.Q THEN
   Bullet_window2:=TRUE ;
END_IF
  
 Bounce_TON(IN:= , PT:=(UDINT_TO_TIME(P3User2_Par.Bounce_time*1000)) , Q=> , ET=> );
 Status_switching_TON(IN:= , PT:=(UDINT_TO_TIME(P3User2_Par.Status_switching_time*1000)) , Q=> , ET=> );
 Status_switching2_TON(IN:= , PT:=(UDINT_TO_TIME(P3User2_Par.Status_switching_time*1000)) , Q=> , ET=> );
 Standby_TON(IN:=(Manual_click_code=6) , PT:=(UDINT_TO_TIME(P3User2_Par.Standby_time*1000)) , Q=> , ET=> );

 
IF Bullet_window2 THEN
   Bounce_TON.IN:=TRUE ;
ELSE
   Bounce_TON.IN:=FALSE ;
END_IF

IF Bounce_TON.Q  THEN
   Bullet_window:=TRUE ;//弹窗触发
   Bullet_window2 :=FALSE ;
  
END_IF
 
IF P3Press.Make_sure THEN
   Bullet_window:=FALSE ;//弹窗关闭
   P3Press.Make_sure:=FALSE ;
END_IF
 
//设备状态
IF P2Btn.P2M1_Tricolorlamp_Green OR P2Btn.P2M2_Tricolorlamp_Green OR P2Btn.P2M3_Tricolorlamp_Green THEN
	 P3Press.Device_Status_code:=7 ; //设备自动中
	 Status_switching_TON.IN:=FALSE ;
	 Status_switching2_TON.IN:=FALSE ;
END_IF

IF ((P2Btn.P2M1_Tricolorlamp_Red AND P2Btn.P2M2_Tricolorlamp_Red AND P2Btn.P2M3_Tricolorlamp_Red  ) OR 
   ((P2M1_DTSysState.bErrorStop OR P2M1_WJSysState.bErrorStop OR P2M1_WJSysState.bErrorStop) AND 
    (P2M2_DTSysState.bErrorStop OR P2M2_WJSysState.bErrorStop OR P2M2_WJSysState.bErrorStop) AND 
   (P2M3_DTSysState.bErrorStop OR P2M3_WJSysState.bErrorStop OR P2M3_WJSysState.bErrorStop)) OR
((P2M1_DTSysState.bErrorStop OR P2M1_WJSysState.bErrorStop OR P2M1_WJSysState.bErrorStop) AND (P2M2_DTSysState.bErrorStop OR P2M2_WJSysState.bErrorStop OR P2M2_WJSysState.bErrorStop)) OR
((P2M1_DTSysState.bErrorStop OR P2M1_WJSysState.bErrorStop OR P2M1_WJSysState.bErrorStop) AND (P2M3_DTSysState.bErrorStop OR P2M3_WJSysState.bErrorStop OR P2M3_WJSysState.bErrorStop)) OR
((P2M2_DTSysState.bErrorStop OR P2M2_WJSysState.bErrorStop OR P2M2_WJSysState.bErrorStop) AND (P2M3_DTSysState.bErrorStop OR P2M3_WJSysState.bErrorStop OR P2M3_WJSysState.bErrorStop))) AND
NOT P2Btn.P2M1_Tricolorlamp_Green AND NOT P2Btn.P2M2_Tricolorlamp_Green AND NOT P2Btn.P2M3_Tricolorlamp_Green AND Manual_click_code<>6  THEN
     Status_switching_TON.IN:=TRUE ;
	 Status_switching2_TON.IN:=FALSE ;
END_IF

IF  Status_switching_TON.Q THEN 
   P3Press.Device_Status_code:=9 ; //设备故障
  
END_IF

